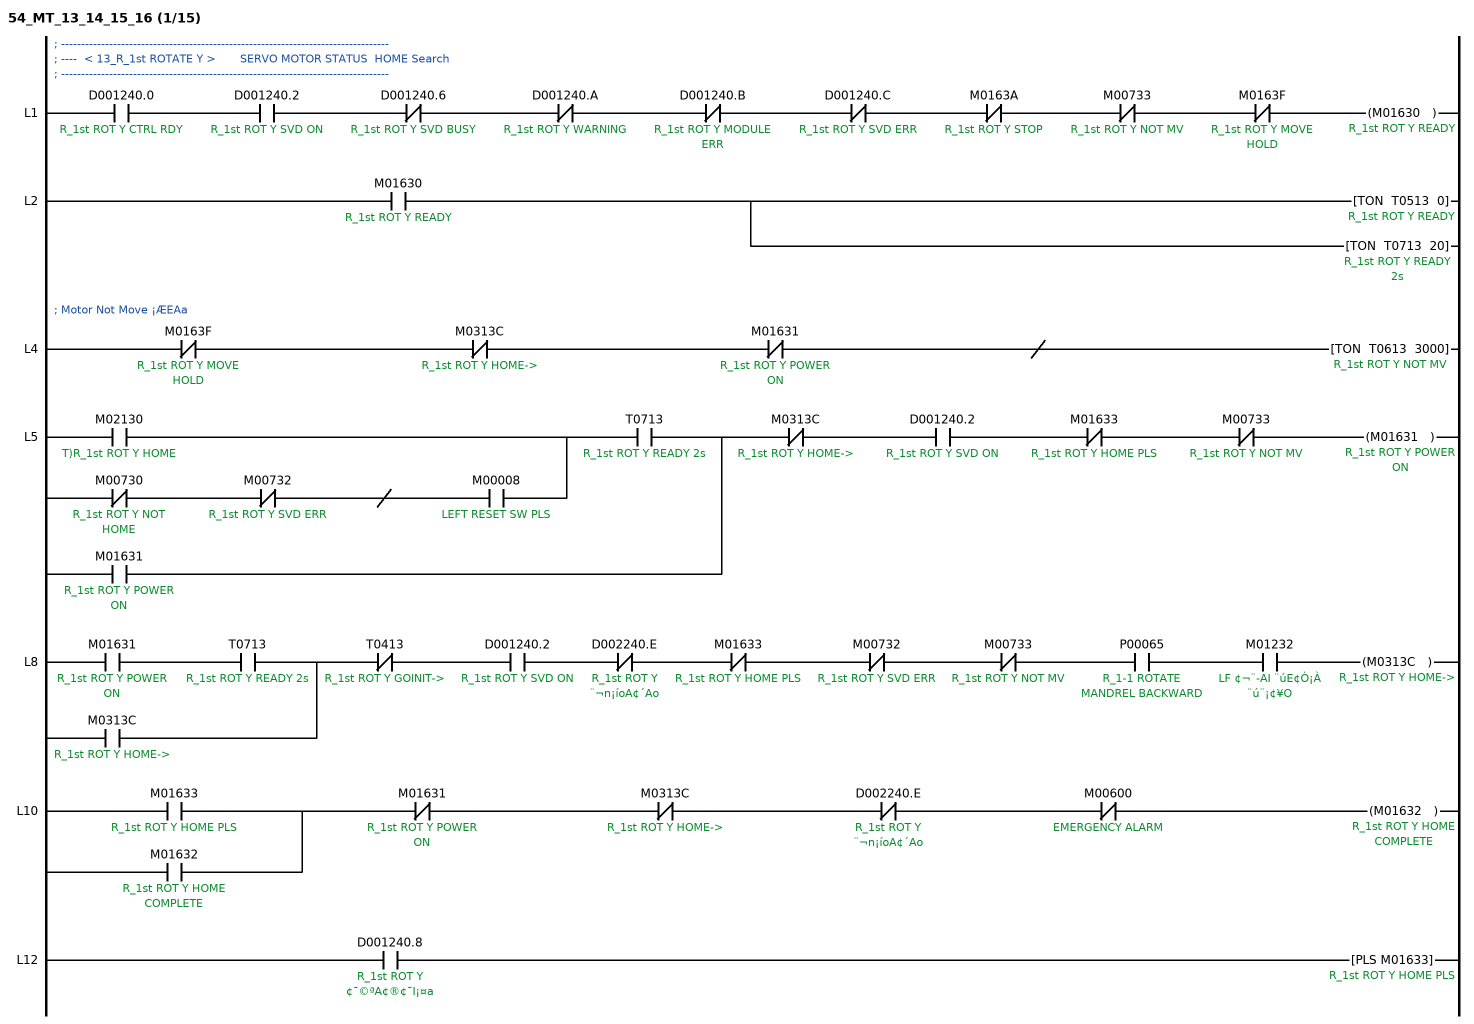
[picture p288: 54_MT_13_14_15_16 rungs L1-L12]
// ----------------------------------------------------------------------------------
// 
// ----  < 13_R_1st ROTATE Y >       SERVO MOTOR STATUS  HOME Search
// 
// ----------------------------------------------------------------------------------
; L1
LOAD      D001240.0	// R_1st ROT Y CTRL RDY
AND       D001240.2	// R_1st ROT Y SVD ON
AND NOT   D001240.6	// R_1st ROT Y SVD BUSY
AND NOT   D001240.A	// R_1st ROT Y WARNING
AND NOT   D001240.B	// R_1st ROT Y MODULE ERR
AND NOT   D001240.C	// R_1st ROT Y SVD ERR
AND NOT   M0163A	// R_1st ROT Y STOP
AND NOT   M00733	// R_1st ROT Y NOT MV
AND NOT   M0163F	// R_1st ROT Y MOVE HOLD
OUT       M01630	// R_1st ROT Y READY
; L2
LOAD      M01630	// R_1st ROT Y READY
TON       T0513 0	// R_1st ROT Y READY
TON       T0713 20	// R_1st ROT Y READY 2s
; L4
LOAD NOT  M0163F	// R_1st ROT Y MOVE HOLD
AND NOT   M0313C	// R_1st ROT Y HOME->
AND NOT   M01631	// R_1st ROT Y POWER ON
NOT
TON       T0613 3000	// R_1st ROT Y NOT MV
// output comment: Motor Not Move ¡ÆEAa
; L5
LOAD      M02130	// T)R_1st ROT Y HOME
LOAD NOT  M00730	// R_1st ROT Y NOT HOME
AND NOT   M00732	// R_1st ROT Y SVD ERR
NOT
AND       M00008	// LEFT RESET SW PLS
OR LOAD
AND       T0713	// R_1st ROT Y READY 2s
OR        M01631	// R_1st ROT Y POWER ON
AND NOT   M0313C	// R_1st ROT Y HOME->
AND       D001240.2	// R_1st ROT Y SVD ON
AND NOT   M01633	// R_1st ROT Y HOME PLS
AND NOT   M00733	// R_1st ROT Y NOT MV
OUT       M01631	// R_1st ROT Y POWER ON
; L8
LOAD      M01631	// R_1st ROT Y POWER ON
AND       T0713	// R_1st ROT Y READY 2s
OR        M0313C	// R_1st ROT Y HOME->
AND NOT   T0413	// R_1st ROT Y GOINIT->
AND       D001240.2	// R_1st ROT Y SVD ON
AND NOT   D002240.E	// R_1st ROT Y ¨¬n¡íoA¢´Ao
AND NOT   M01633	// R_1st ROT Y HOME PLS
AND NOT   M00732	// R_1st ROT Y SVD ERR
AND NOT   M00733	// R_1st ROT Y NOT MV
AND       P00065	// R_1-1 ROTATE MANDREL BACKWARD
AND       M01232	// LF ¢¬¨­AI ¨úE¢Ò¡À ¨ú¨¡¢¥O
OUT       M0313C	// R_1st ROT Y HOME->
; L10
LOAD      M01633	// R_1st ROT Y HOME PLS
OR        M01632	// R_1st ROT Y HOME COMPLETE
AND NOT   M01631	// R_1st ROT Y POWER ON
AND NOT   M0313C	// R_1st ROT Y HOME->
AND NOT   D002240.E	// R_1st ROT Y ¨¬n¡íoA¢´Ao
AND NOT   M00600	// EMERGENCY ALARM
OUT       M01632	// R_1st ROT Y HOME COMPLETE
; L12
LOAD      D001240.8	// R_1st ROT Y ¢¯©ªA¢®¢¯I¡¤a
OUTP      M01633	// R_1st ROT Y HOME PLS

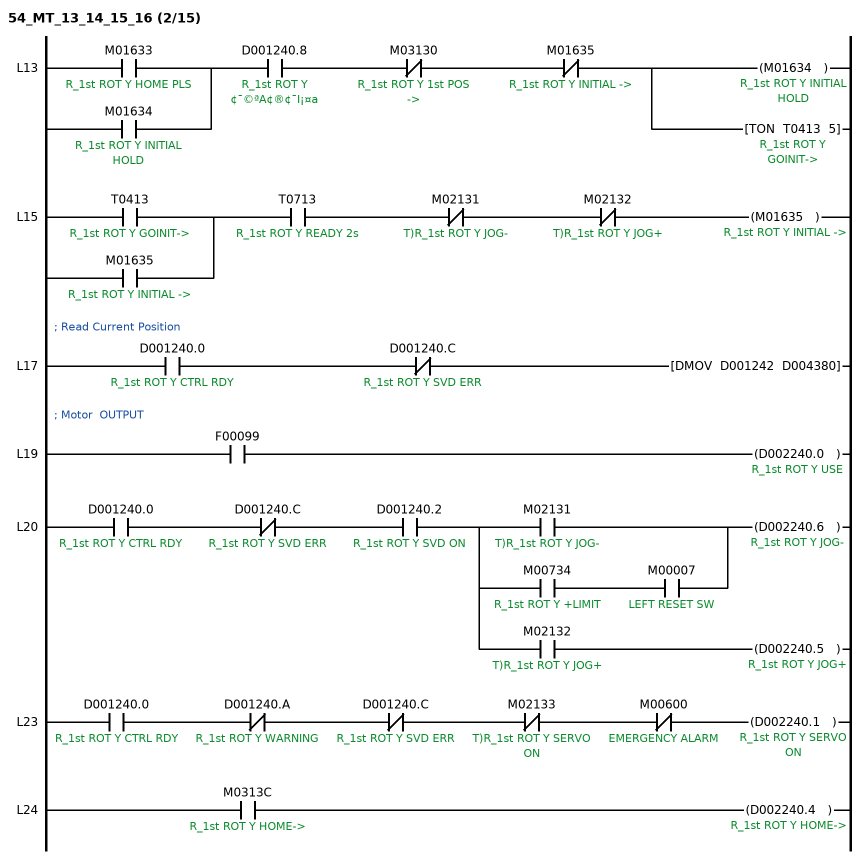
; L13
LOAD      M01633	// R_1st ROT Y HOME PLS
OR        M01634	// R_1st ROT Y INITIAL HOLD
AND       D001240.8	// R_1st ROT Y ¢¯©ªA¢®¢¯I¡¤a
AND NOT   M03130	// R_1st ROT Y 1st POS ->
AND NOT   M01635	// R_1st ROT Y INITIAL ->
OUT       M01634	// R_1st ROT Y INITIAL HOLD
TON       T0413 5	// R_1st ROT Y GOINIT->
; L15
LOAD      T0413	// R_1st ROT Y GOINIT->
OR        M01635	// R_1st ROT Y INITIAL ->
AND       T0713	// R_1st ROT Y READY 2s
AND NOT   M02131	// T)R_1st ROT Y JOG-
AND NOT   M02132	// T)R_1st ROT Y JOG+
OUT       M01635	// R_1st ROT Y INITIAL ->
; L17
LOAD      D001240.0	// R_1st ROT Y CTRL RDY
AND NOT   D001240.C	// R_1st ROT Y SVD ERR
DMOV      D001242 D004380
// output comment: Read Current Position
//  Motor  OUTPUT
; L19
LOAD      F00099
OUT       D002240.0	// R_1st ROT Y USE
; L20
LOAD      D001240.0	// R_1st ROT Y CTRL RDY
AND NOT   D001240.C	// R_1st ROT Y SVD ERR
AND       D001240.2	// R_1st ROT Y SVD ON
MPUSH
LOAD      M02131	// T)R_1st ROT Y JOG-
LOAD      M00734	// R_1st ROT Y +LIMIT
AND       M00007	// LEFT RESET SW
OR LOAD
AND LOAD
OUT       D002240.6	// R_1st ROT Y JOG-
MPOP
AND       M02132	// T)R_1st ROT Y JOG+
OUT       D002240.5	// R_1st ROT Y JOG+
; L23
LOAD      D001240.0	// R_1st ROT Y CTRL RDY
AND NOT   D001240.A	// R_1st ROT Y WARNING
AND NOT   D001240.C	// R_1st ROT Y SVD ERR
AND NOT   M02133	// T)R_1st ROT Y SERVO ON
AND NOT   M00600	// EMERGENCY ALARM
OUT       D002240.1	// R_1st ROT Y SERVO ON
; L24
LOAD      M0313C	// R_1st ROT Y HOME->
OUT       D002240.4	// R_1st ROT Y HOME->

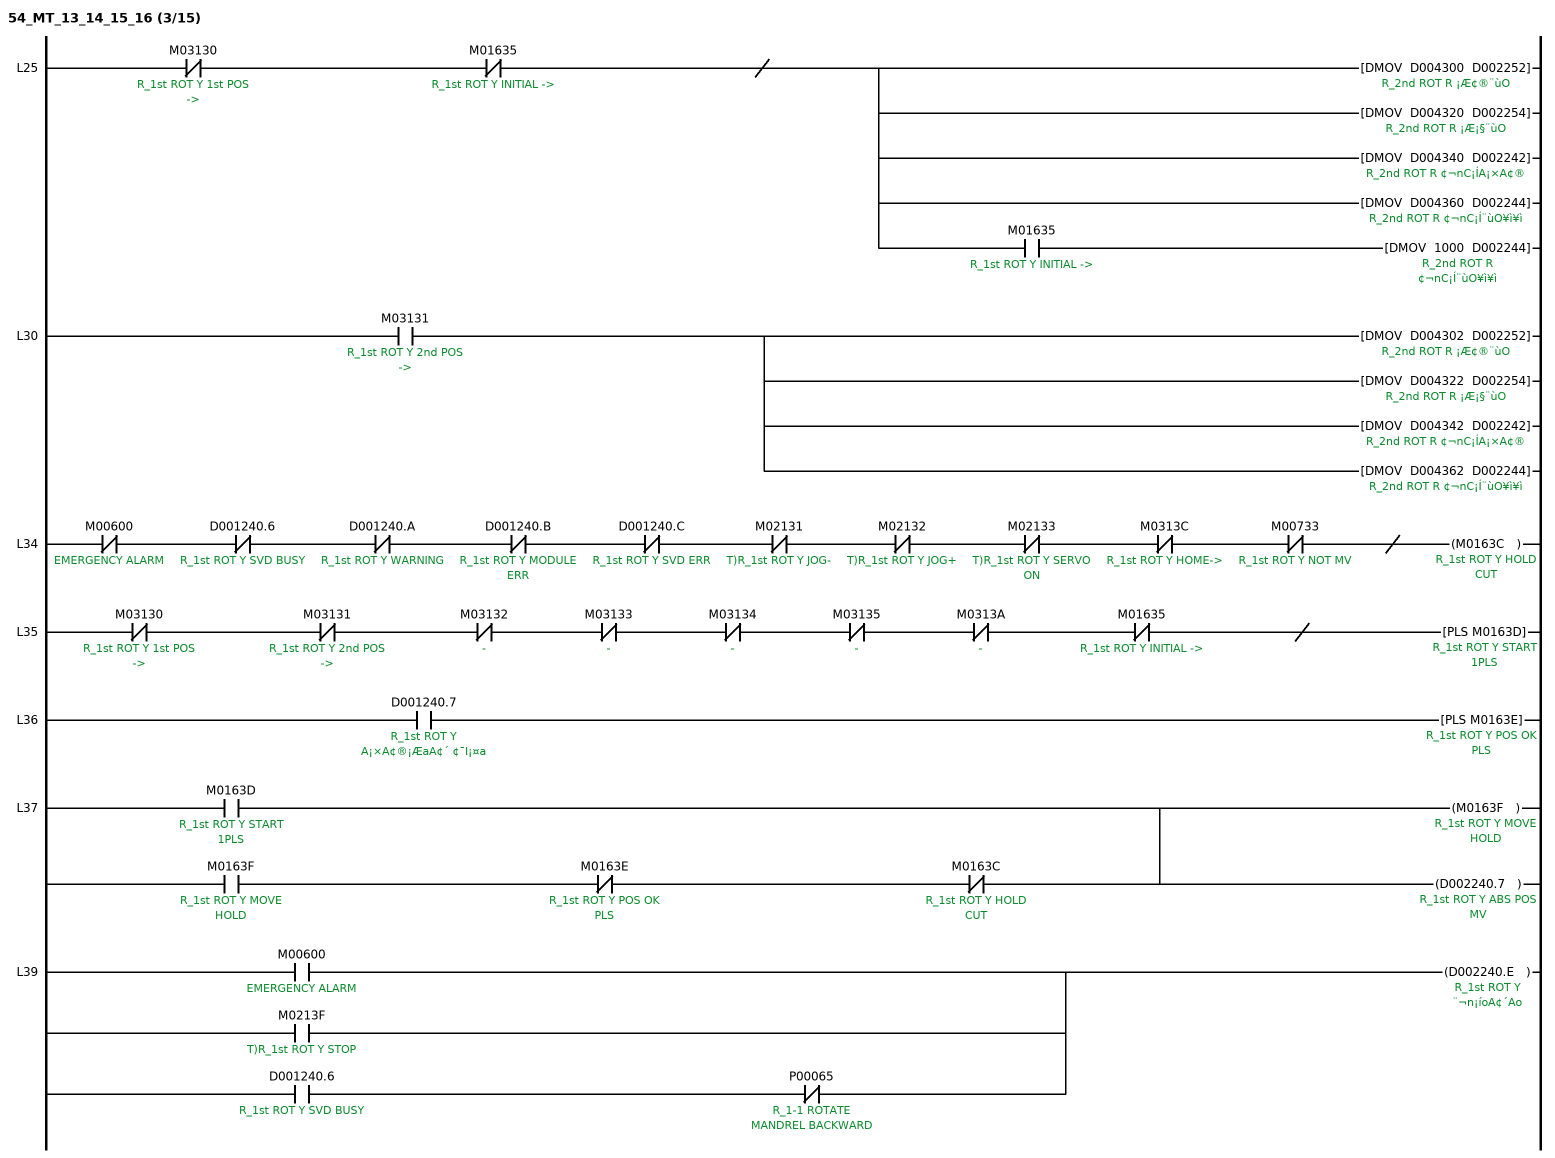
; L25
LOAD NOT  M03130	// R_1st ROT Y 1st POS ->
AND NOT   M01635	// R_1st ROT Y INITIAL ->
NOT
DMOV      D004300 D002252	// R_2nd ROT R ¡Æ¢®¨ùO
DMOV      D004320 D002254	// R_2nd ROT R ¡Æ¡§¨ùO
DMOV      D004340 D002242	// R_2nd ROT R ¢¬nC¡ÍA¡×A¢®
DMOV      D004360 D002244	// R_2nd ROT R ¢¬nC¡Í¨ùO¥ì¥ì
AND       M01635	// R_1st ROT Y INITIAL ->
DMOV      1000 D002244	// R_2nd ROT R ¢¬nC¡Í¨ùO¥ì¥ì
; L30
LOAD      M03131	// R_1st ROT Y 2nd POS ->
DMOV      D004302 D002252	// R_2nd ROT R ¡Æ¢®¨ùO
DMOV      D004322 D002254	// R_2nd ROT R ¡Æ¡§¨ùO
DMOV      D004342 D002242	// R_2nd ROT R ¢¬nC¡ÍA¡×A¢®
DMOV      D004362 D002244	// R_2nd ROT R ¢¬nC¡Í¨ùO¥ì¥ì
; L34
LOAD NOT  M00600	// EMERGENCY ALARM
AND NOT   D001240.6	// R_1st ROT Y SVD BUSY
AND NOT   D001240.A	// R_1st ROT Y WARNING
AND NOT   D001240.B	// R_1st ROT Y MODULE ERR
AND NOT   D001240.C	// R_1st ROT Y SVD ERR
AND NOT   M02131	// T)R_1st ROT Y JOG-
AND NOT   M02132	// T)R_1st ROT Y JOG+
AND NOT   M02133	// T)R_1st ROT Y SERVO ON
AND NOT   M0313C	// R_1st ROT Y HOME->
AND NOT   M00733	// R_1st ROT Y NOT MV
NOT
OUT       M0163C	// R_1st ROT Y HOLD CUT
; L35
LOAD NOT  M03130	// R_1st ROT Y 1st POS ->
AND NOT   M03131	// R_1st ROT Y 2nd POS ->
AND NOT   M03132	// -
AND NOT   M03133	// -
AND NOT   M03134	// -
AND NOT   M03135	// -
AND NOT   M0313A	// -
AND NOT   M01635	// R_1st ROT Y INITIAL ->
NOT
OUTP      M0163D	// R_1st ROT Y START 1PLS
; L36
LOAD      D001240.7	// R_1st ROT Y A¡×A¢®¡ÆaA¢´ ¢¯I¡¤a
OUTP      M0163E	// R_1st ROT Y POS OK PLS
; L37
LOAD      M0163D	// R_1st ROT Y START 1PLS
LOAD      M0163F	// R_1st ROT Y MOVE HOLD
AND NOT   M0163E	// R_1st ROT Y POS OK PLS
AND NOT   M0163C	// R_1st ROT Y HOLD CUT
OR LOAD
OUT       M0163F	// R_1st ROT Y MOVE HOLD
OUT       D002240.7	// R_1st ROT Y ABS POS MV
; L39
LOAD      M00600	// EMERGENCY ALARM
OR        M0213F	// T)R_1st ROT Y STOP
LOAD      D001240.6	// R_1st ROT Y SVD BUSY
AND NOT   P00065	// R_1-1 ROTATE MANDREL BACKWARD
OR LOAD
OUT       D002240.E	// R_1st ROT Y ¨¬n¡íoA¢´Ao

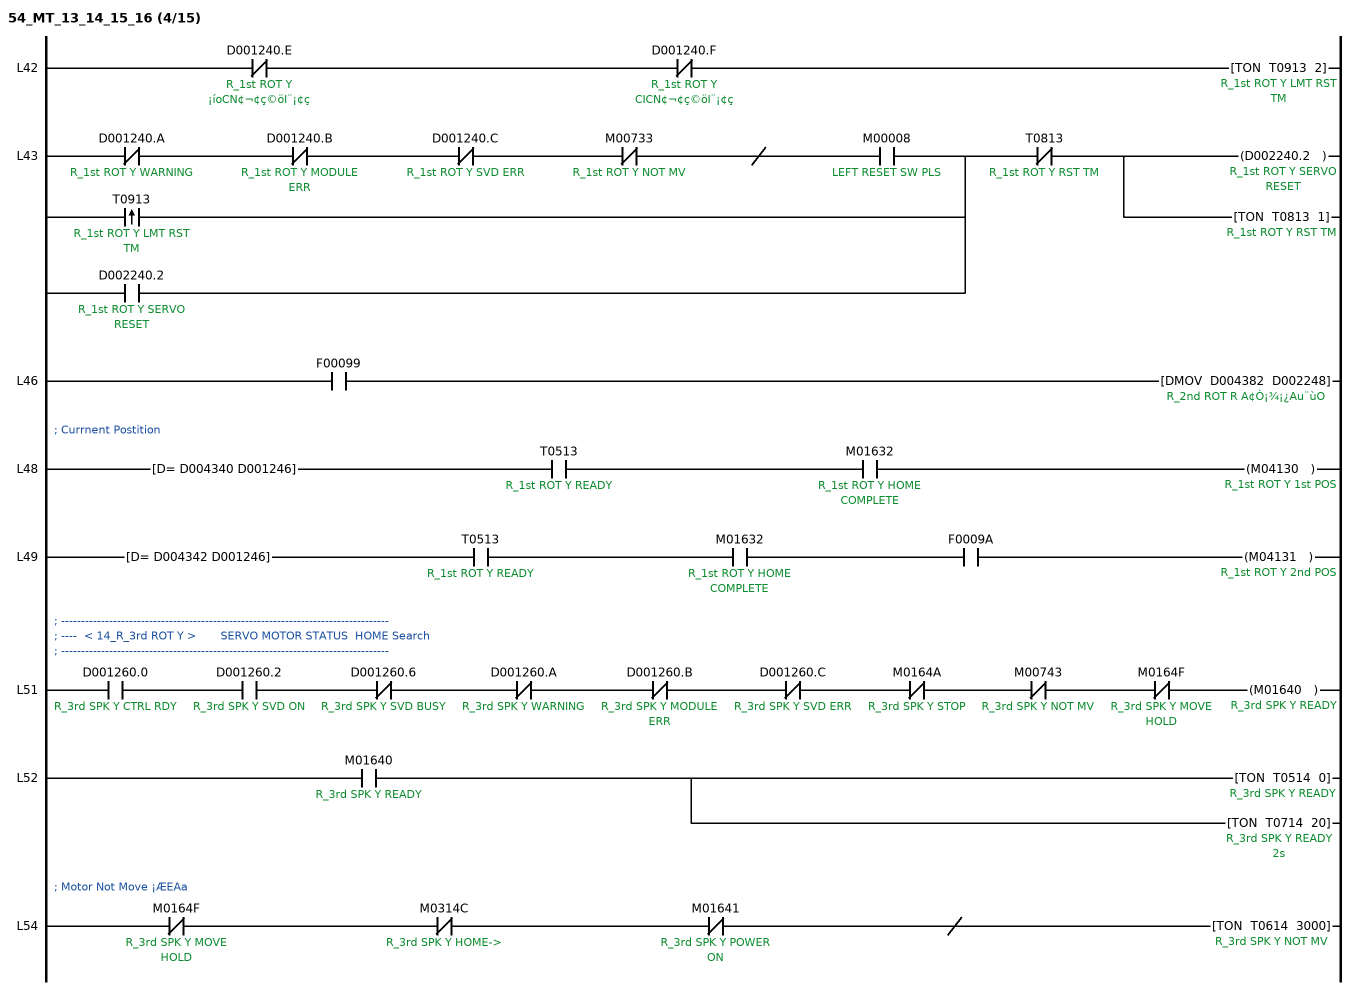
; L42
LOAD NOT  D001240.E	// R_1st ROT Y ¡íoCN¢¬¢ç©öI¨¡¢ç
AND NOT   D001240.F	// R_1st ROT Y CICN¢¬¢ç©öI¨¡¢ç
TON       T0913 2	// R_1st ROT Y LMT RST TM
; L43
LOAD NOT  D001240.A	// R_1st ROT Y WARNING
AND NOT   D001240.B	// R_1st ROT Y MODULE ERR
AND NOT   D001240.C	// R_1st ROT Y SVD ERR
AND NOT   M00733	// R_1st ROT Y NOT MV
NOT
AND       M00008	// LEFT RESET SW PLS
ORP       T0913	// R_1st ROT Y LMT RST TM
OR        D002240.2	// R_1st ROT Y SERVO RESET
AND NOT   T0813	// R_1st ROT Y RST TM
OUT       D002240.2	// R_1st ROT Y SERVO RESET
TON       T0813 1	// R_1st ROT Y RST TM
; L46
LOAD      F00099
DMOV      D004382 D002248	// R_2nd ROT R A¢Ò¡¾¡¿Au¨ùO
// Currnent Postition
; L48
LOADD=    D004340 D001246
AND       T0513	// R_1st ROT Y READY
AND       M01632	// R_1st ROT Y HOME COMPLETE
OUT       M04130	// R_1st ROT Y 1st POS
; L49
LOADD=    D004342 D001246
AND       T0513	// R_1st ROT Y READY
AND       M01632	// R_1st ROT Y HOME COMPLETE
AND       F0009A
OUT       M04131	// R_1st ROT Y 2nd POS
// ----------------------------------------------------------------------------------
// 
// ----  < 14_R_3rd ROT Y >       SERVO MOTOR STATUS  HOME Search
// 
// ----------------------------------------------------------------------------------
; L51
LOAD      D001260.0	// R_3rd SPK Y CTRL RDY
AND       D001260.2	// R_3rd SPK Y SVD ON
AND NOT   D001260.6	// R_3rd SPK Y SVD BUSY
AND NOT   D001260.A	// R_3rd SPK Y WARNING
AND NOT   D001260.B	// R_3rd SPK Y MODULE ERR
AND NOT   D001260.C	// R_3rd SPK Y SVD ERR
AND NOT   M0164A	// R_3rd SPK Y STOP
AND NOT   M00743	// R_3rd SPK Y NOT MV
AND NOT   M0164F	// R_3rd SPK Y MOVE HOLD
OUT       M01640	// R_3rd SPK Y READY
; L52
LOAD      M01640	// R_3rd SPK Y READY
TON       T0514 0	// R_3rd SPK Y READY
TON       T0714 20	// R_3rd SPK Y READY 2s
; L54
LOAD NOT  M0164F	// R_3rd SPK Y MOVE HOLD
AND NOT   M0314C	// R_3rd SPK Y HOME->
AND NOT   M01641	// R_3rd SPK Y POWER ON
NOT
TON       T0614 3000	// R_3rd SPK Y NOT MV
// output comment: Motor Not Move ¡ÆEAa

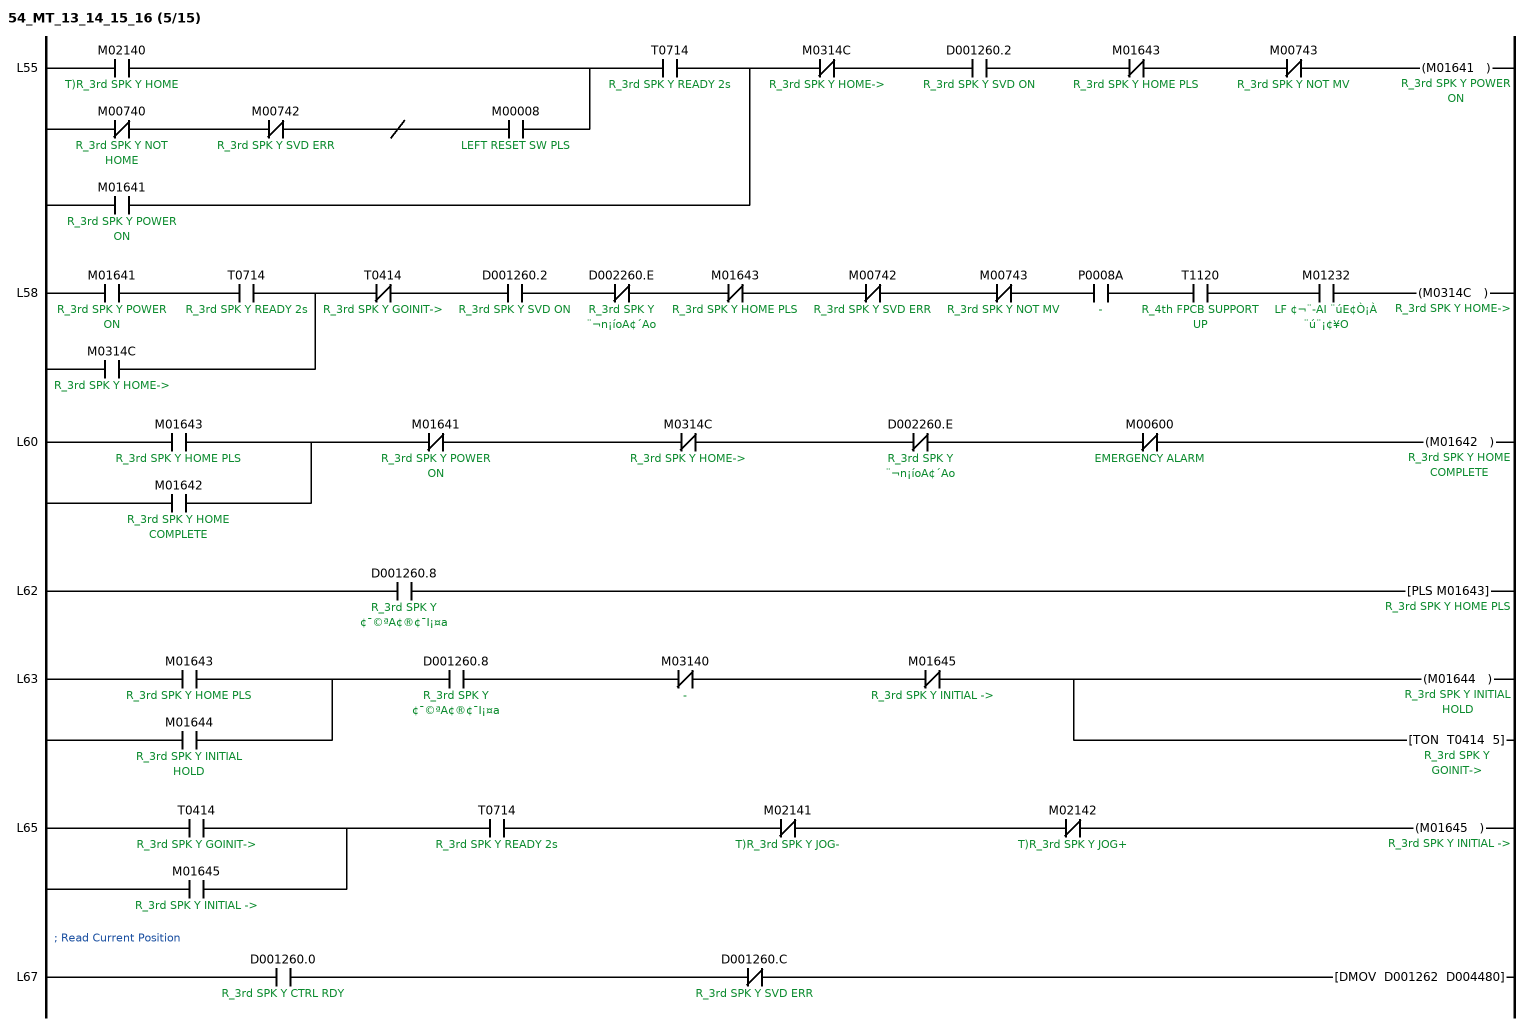
; L55
LOAD      M02140	// T)R_3rd SPK Y HOME
LOAD NOT  M00740	// R_3rd SPK Y NOT HOME
AND NOT   M00742	// R_3rd SPK Y SVD ERR
NOT
AND       M00008	// LEFT RESET SW PLS
OR LOAD
AND       T0714	// R_3rd SPK Y READY 2s
OR        M01641	// R_3rd SPK Y POWER ON
AND NOT   M0314C	// R_3rd SPK Y HOME->
AND       D001260.2	// R_3rd SPK Y SVD ON
AND NOT   M01643	// R_3rd SPK Y HOME PLS
AND NOT   M00743	// R_3rd SPK Y NOT MV
OUT       M01641	// R_3rd SPK Y POWER ON
; L58
LOAD      M01641	// R_3rd SPK Y POWER ON
AND       T0714	// R_3rd SPK Y READY 2s
OR        M0314C	// R_3rd SPK Y HOME->
AND NOT   T0414	// R_3rd SPK Y GOINIT->
AND       D001260.2	// R_3rd SPK Y SVD ON
AND NOT   D002260.E	// R_3rd SPK Y ¨¬n¡íoA¢´Ao
AND NOT   M01643	// R_3rd SPK Y HOME PLS
AND NOT   M00742	// R_3rd SPK Y SVD ERR
AND NOT   M00743	// R_3rd SPK Y NOT MV
AND       P0008A	// -
AND       T1120	// R_4th FPCB SUPPORT UP
AND       M01232	// LF ¢¬¨­AI ¨úE¢Ò¡À ¨ú¨¡¢¥O
OUT       M0314C	// R_3rd SPK Y HOME->
; L60
LOAD      M01643	// R_3rd SPK Y HOME PLS
OR        M01642	// R_3rd SPK Y HOME COMPLETE
AND NOT   M01641	// R_3rd SPK Y POWER ON
AND NOT   M0314C	// R_3rd SPK Y HOME->
AND NOT   D002260.E	// R_3rd SPK Y ¨¬n¡íoA¢´Ao
AND NOT   M00600	// EMERGENCY ALARM
OUT       M01642	// R_3rd SPK Y HOME COMPLETE
; L62
LOAD      D001260.8	// R_3rd SPK Y ¢¯©ªA¢®¢¯I¡¤a
OUTP      M01643	// R_3rd SPK Y HOME PLS
; L63
LOAD      M01643	// R_3rd SPK Y HOME PLS
OR        M01644	// R_3rd SPK Y INITIAL HOLD
AND       D001260.8	// R_3rd SPK Y ¢¯©ªA¢®¢¯I¡¤a
AND NOT   M03140	// -
AND NOT   M01645	// R_3rd SPK Y INITIAL ->
OUT       M01644	// R_3rd SPK Y INITIAL HOLD
TON       T0414 5	// R_3rd SPK Y GOINIT->
; L65
LOAD      T0414	// R_3rd SPK Y GOINIT->
OR        M01645	// R_3rd SPK Y INITIAL ->
AND       T0714	// R_3rd SPK Y READY 2s
AND NOT   M02141	// T)R_3rd SPK Y JOG-
AND NOT   M02142	// T)R_3rd SPK Y JOG+
OUT       M01645	// R_3rd SPK Y INITIAL ->
; L67
LOAD      D001260.0	// R_3rd SPK Y CTRL RDY
AND NOT   D001260.C	// R_3rd SPK Y SVD ERR
DMOV      D001262 D004480
// output comment: Read Current Position

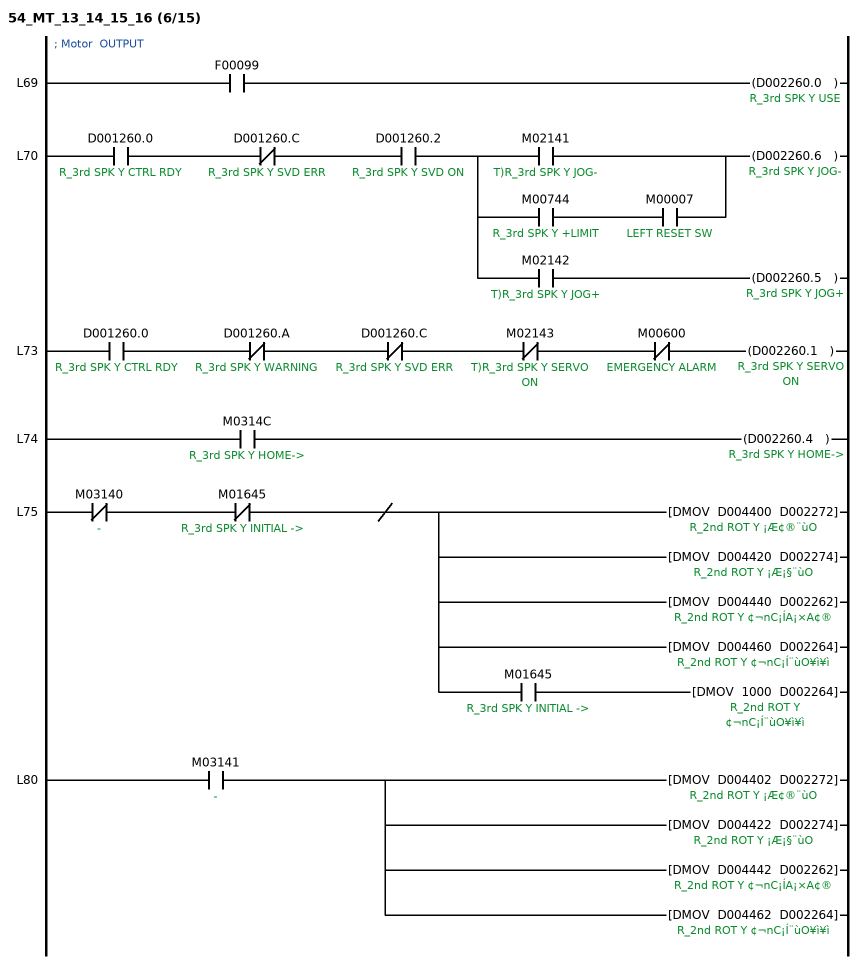
//  Motor  OUTPUT
; L69
LOAD      F00099
OUT       D002260.0	// R_3rd SPK Y USE
; L70
LOAD      D001260.0	// R_3rd SPK Y CTRL RDY
AND NOT   D001260.C	// R_3rd SPK Y SVD ERR
AND       D001260.2	// R_3rd SPK Y SVD ON
MPUSH
LOAD      M02141	// T)R_3rd SPK Y JOG-
LOAD      M00744	// R_3rd SPK Y +LIMIT
AND       M00007	// LEFT RESET SW
OR LOAD
AND LOAD
OUT       D002260.6	// R_3rd SPK Y JOG-
MPOP
AND       M02142	// T)R_3rd SPK Y JOG+
OUT       D002260.5	// R_3rd SPK Y JOG+
; L73
LOAD      D001260.0	// R_3rd SPK Y CTRL RDY
AND NOT   D001260.A	// R_3rd SPK Y WARNING
AND NOT   D001260.C	// R_3rd SPK Y SVD ERR
AND NOT   M02143	// T)R_3rd SPK Y SERVO ON
AND NOT   M00600	// EMERGENCY ALARM
OUT       D002260.1	// R_3rd SPK Y SERVO ON
; L74
LOAD      M0314C	// R_3rd SPK Y HOME->
OUT       D002260.4	// R_3rd SPK Y HOME->
; L75
LOAD NOT  M03140	// -
AND NOT   M01645	// R_3rd SPK Y INITIAL ->
NOT
DMOV      D004400 D002272	// R_2nd ROT Y ¡Æ¢®¨ùO
DMOV      D004420 D002274	// R_2nd ROT Y ¡Æ¡§¨ùO
DMOV      D004440 D002262	// R_2nd ROT Y ¢¬nC¡ÍA¡×A¢®
DMOV      D004460 D002264	// R_2nd ROT Y ¢¬nC¡Í¨ùO¥ì¥ì
AND       M01645	// R_3rd SPK Y INITIAL ->
DMOV      1000 D002264	// R_2nd ROT Y ¢¬nC¡Í¨ùO¥ì¥ì
; L80
LOAD      M03141	// -
DMOV      D004402 D002272	// R_2nd ROT Y ¡Æ¢®¨ùO
DMOV      D004422 D002274	// R_2nd ROT Y ¡Æ¡§¨ùO
DMOV      D004442 D002262	// R_2nd ROT Y ¢¬nC¡ÍA¡×A¢®
DMOV      D004462 D002264	// R_2nd ROT Y ¢¬nC¡Í¨ùO¥ì¥ì

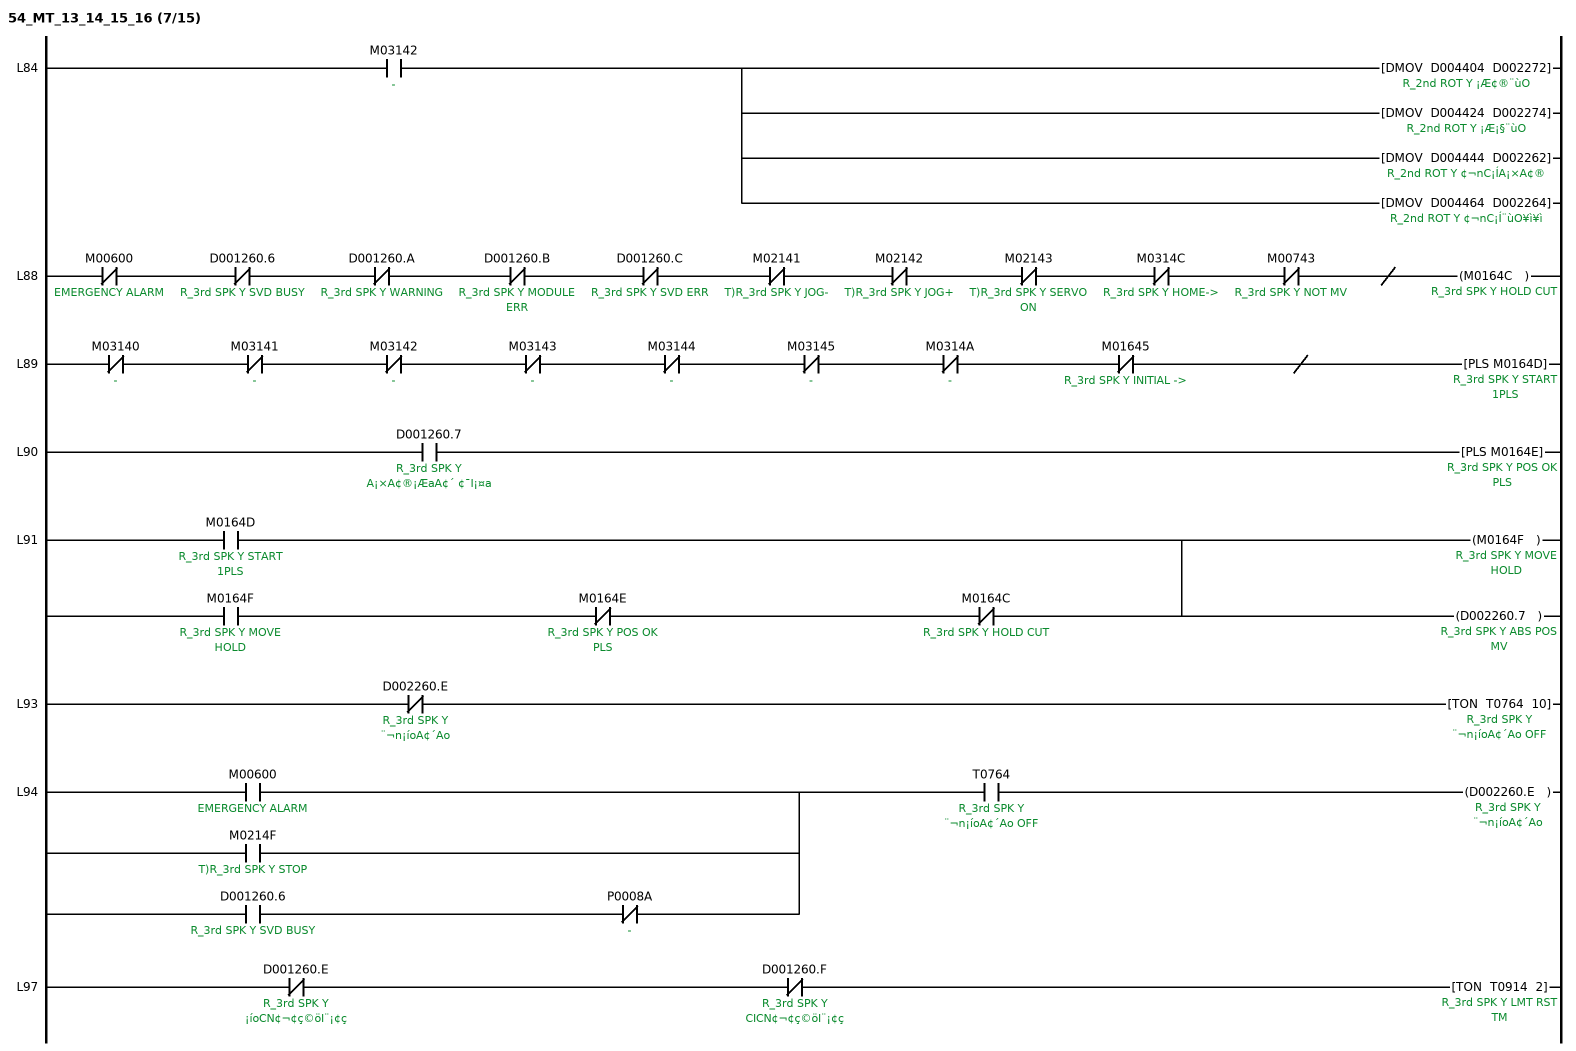
; L84
LOAD      M03142	// -
DMOV      D004404 D002272	// R_2nd ROT Y ¡Æ¢®¨ùO
DMOV      D004424 D002274	// R_2nd ROT Y ¡Æ¡§¨ùO
DMOV      D004444 D002262	// R_2nd ROT Y ¢¬nC¡ÍA¡×A¢®
DMOV      D004464 D002264	// R_2nd ROT Y ¢¬nC¡Í¨ùO¥ì¥ì
; L88
LOAD NOT  M00600	// EMERGENCY ALARM
AND NOT   D001260.6	// R_3rd SPK Y SVD BUSY
AND NOT   D001260.A	// R_3rd SPK Y WARNING
AND NOT   D001260.B	// R_3rd SPK Y MODULE ERR
AND NOT   D001260.C	// R_3rd SPK Y SVD ERR
AND NOT   M02141	// T)R_3rd SPK Y JOG-
AND NOT   M02142	// T)R_3rd SPK Y JOG+
AND NOT   M02143	// T)R_3rd SPK Y SERVO ON
AND NOT   M0314C	// R_3rd SPK Y HOME->
AND NOT   M00743	// R_3rd SPK Y NOT MV
NOT
OUT       M0164C	// R_3rd SPK Y HOLD CUT
; L89
LOAD NOT  M03140	// -
AND NOT   M03141	// -
AND NOT   M03142	// -
AND NOT   M03143	// -
AND NOT   M03144	// -
AND NOT   M03145	// -
AND NOT   M0314A	// -
AND NOT   M01645	// R_3rd SPK Y INITIAL ->
NOT
OUTP      M0164D	// R_3rd SPK Y START 1PLS
; L90
LOAD      D001260.7	// R_3rd SPK Y A¡×A¢®¡ÆaA¢´ ¢¯I¡¤a
OUTP      M0164E	// R_3rd SPK Y POS OK PLS
; L91
LOAD      M0164D	// R_3rd SPK Y START 1PLS
LOAD      M0164F	// R_3rd SPK Y MOVE HOLD
AND NOT   M0164E	// R_3rd SPK Y POS OK PLS
AND NOT   M0164C	// R_3rd SPK Y HOLD CUT
OR LOAD
OUT       M0164F	// R_3rd SPK Y MOVE HOLD
OUT       D002260.7	// R_3rd SPK Y ABS POS MV
; L93
LOAD NOT  D002260.E	// R_3rd SPK Y ¨¬n¡íoA¢´Ao
TON       T0764 10	// R_3rd SPK Y ¨¬n¡íoA¢´Ao OFF
; L94
LOAD      M00600	// EMERGENCY ALARM
OR        M0214F	// T)R_3rd SPK Y STOP
LOAD      D001260.6	// R_3rd SPK Y SVD BUSY
AND NOT   P0008A	// -
OR LOAD
AND       T0764	// R_3rd SPK Y ¨¬n¡íoA¢´Ao OFF
OUT       D002260.E	// R_3rd SPK Y ¨¬n¡íoA¢´Ao
; L97
LOAD NOT  D001260.E	// R_3rd SPK Y ¡íoCN¢¬¢ç©öI¨¡¢ç
AND NOT   D001260.F	// R_3rd SPK Y CICN¢¬¢ç©öI¨¡¢ç
TON       T0914 2	// R_3rd SPK Y LMT RST TM

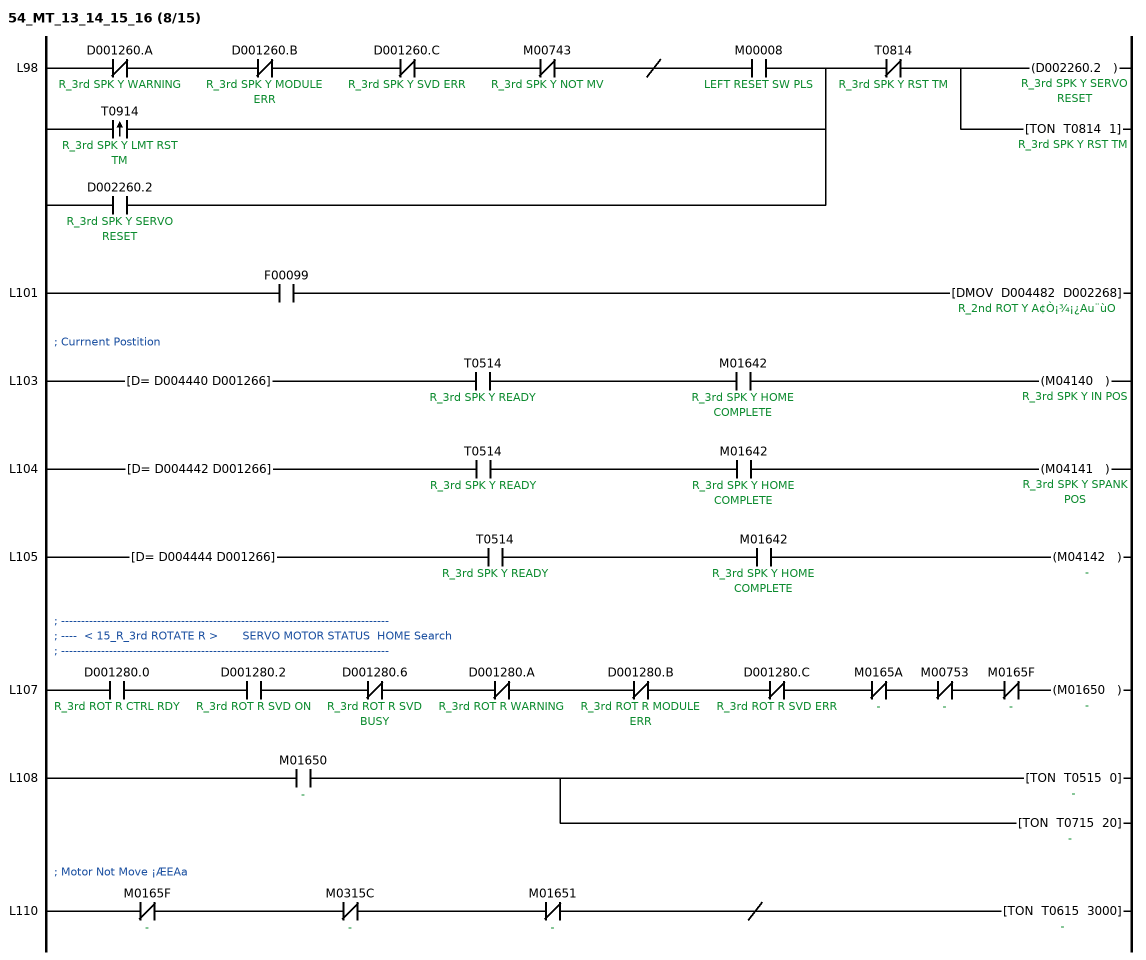
; L98
LOAD NOT  D001260.A	// R_3rd SPK Y WARNING
AND NOT   D001260.B	// R_3rd SPK Y MODULE ERR
AND NOT   D001260.C	// R_3rd SPK Y SVD ERR
AND NOT   M00743	// R_3rd SPK Y NOT MV
NOT
AND       M00008	// LEFT RESET SW PLS
ORP       T0914	// R_3rd SPK Y LMT RST TM
OR        D002260.2	// R_3rd SPK Y SERVO RESET
AND NOT   T0814	// R_3rd SPK Y RST TM
OUT       D002260.2	// R_3rd SPK Y SERVO RESET
TON       T0814 1	// R_3rd SPK Y RST TM
; L101
LOAD      F00099
DMOV      D004482 D002268	// R_2nd ROT Y A¢Ò¡¾¡¿Au¨ùO
// Currnent Postition
; L103
LOADD=    D004440 D001266
AND       T0514	// R_3rd SPK Y READY
AND       M01642	// R_3rd SPK Y HOME COMPLETE
OUT       M04140	// R_3rd SPK Y IN POS
; L104
LOADD=    D004442 D001266
AND       T0514	// R_3rd SPK Y READY
AND       M01642	// R_3rd SPK Y HOME COMPLETE
OUT       M04141	// R_3rd SPK Y SPANK POS
; L105
LOADD=    D004444 D001266
AND       T0514	// R_3rd SPK Y READY
AND       M01642	// R_3rd SPK Y HOME COMPLETE
OUT       M04142	// -
// ----------------------------------------------------------------------------------
// 
// ----  < 15_R_3rd ROTATE R >       SERVO MOTOR STATUS  HOME Search
// 
// ----------------------------------------------------------------------------------
; L107
LOAD      D001280.0	// R_3rd ROT R CTRL RDY
AND       D001280.2	// R_3rd ROT R SVD ON
AND NOT   D001280.6	// R_3rd ROT R SVD BUSY
AND NOT   D001280.A	// R_3rd ROT R WARNING
AND NOT   D001280.B	// R_3rd ROT R MODULE ERR
AND NOT   D001280.C	// R_3rd ROT R SVD ERR
AND NOT   M0165A	// -
AND NOT   M00753	// -
AND NOT   M0165F	// -
OUT       M01650	// -
; L108
LOAD      M01650	// -
TON       T0515 0	// -
TON       T0715 20	// -
; L110
LOAD NOT  M0165F	// -
AND NOT   M0315C	// -
AND NOT   M01651	// -
NOT
TON       T0615 3000	// -
// output comment: Motor Not Move ¡ÆEAa

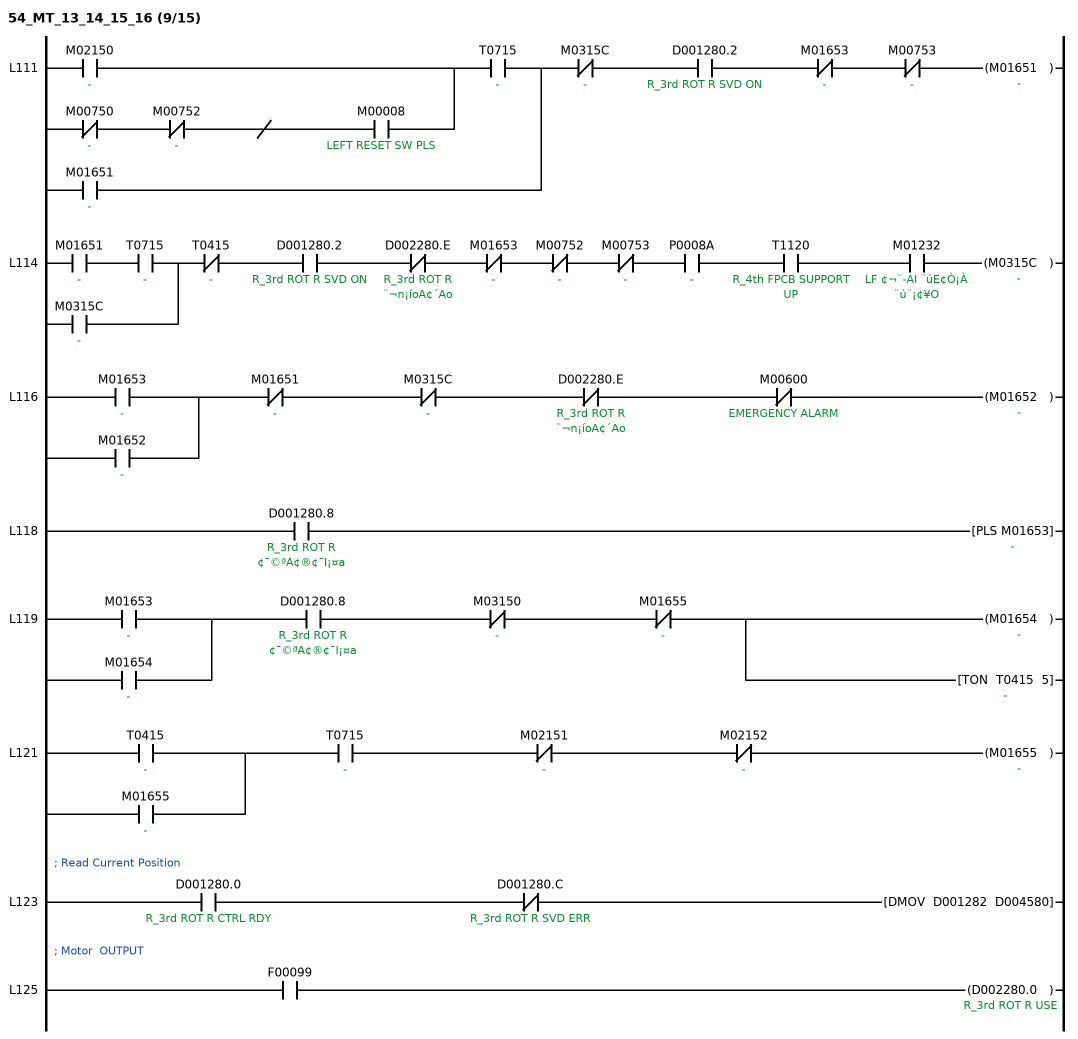
; L111
LOAD      M02150	// -
LOAD NOT  M00750	// -
AND NOT   M00752	// -
NOT
AND       M00008	// LEFT RESET SW PLS
OR LOAD
AND       T0715	// -
OR        M01651	// -
AND NOT   M0315C	// -
AND       D001280.2	// R_3rd ROT R SVD ON
AND NOT   M01653	// -
AND NOT   M00753	// -
OUT       M01651	// -
; L114
LOAD      M01651	// -
AND       T0715	// -
OR        M0315C	// -
AND NOT   T0415	// -
AND       D001280.2	// R_3rd ROT R SVD ON
AND NOT   D002280.E	// R_3rd ROT R ¨¬n¡íoA¢´Ao
AND NOT   M01653	// -
AND NOT   M00752	// -
AND NOT   M00753	// -
AND       P0008A	// -
AND       T1120	// R_4th FPCB SUPPORT UP
AND       M01232	// LF ¢¬¨­AI ¨úE¢Ò¡À ¨ú¨¡¢¥O
OUT       M0315C	// -
; L116
LOAD      M01653	// -
OR        M01652	// -
AND NOT   M01651	// -
AND NOT   M0315C	// -
AND NOT   D002280.E	// R_3rd ROT R ¨¬n¡íoA¢´Ao
AND NOT   M00600	// EMERGENCY ALARM
OUT       M01652	// -
; L118
LOAD      D001280.8	// R_3rd ROT R ¢¯©ªA¢®¢¯I¡¤a
OUTP      M01653	// -
; L119
LOAD      M01653	// -
OR        M01654	// -
AND       D001280.8	// R_3rd ROT R ¢¯©ªA¢®¢¯I¡¤a
AND NOT   M03150	// -
AND NOT   M01655	// -
OUT       M01654	// -
TON       T0415 5	// -
; L121
LOAD      T0415	// -
OR        M01655	// -
AND       T0715	// -
AND NOT   M02151	// -
AND NOT   M02152	// -
OUT       M01655	// -
; L123
LOAD      D001280.0	// R_3rd ROT R CTRL RDY
AND NOT   D001280.C	// R_3rd ROT R SVD ERR
DMOV      D001282 D004580
// output comment: Read Current Position
//  Motor  OUTPUT
; L125
LOAD      F00099
OUT       D002280.0	// R_3rd ROT R USE

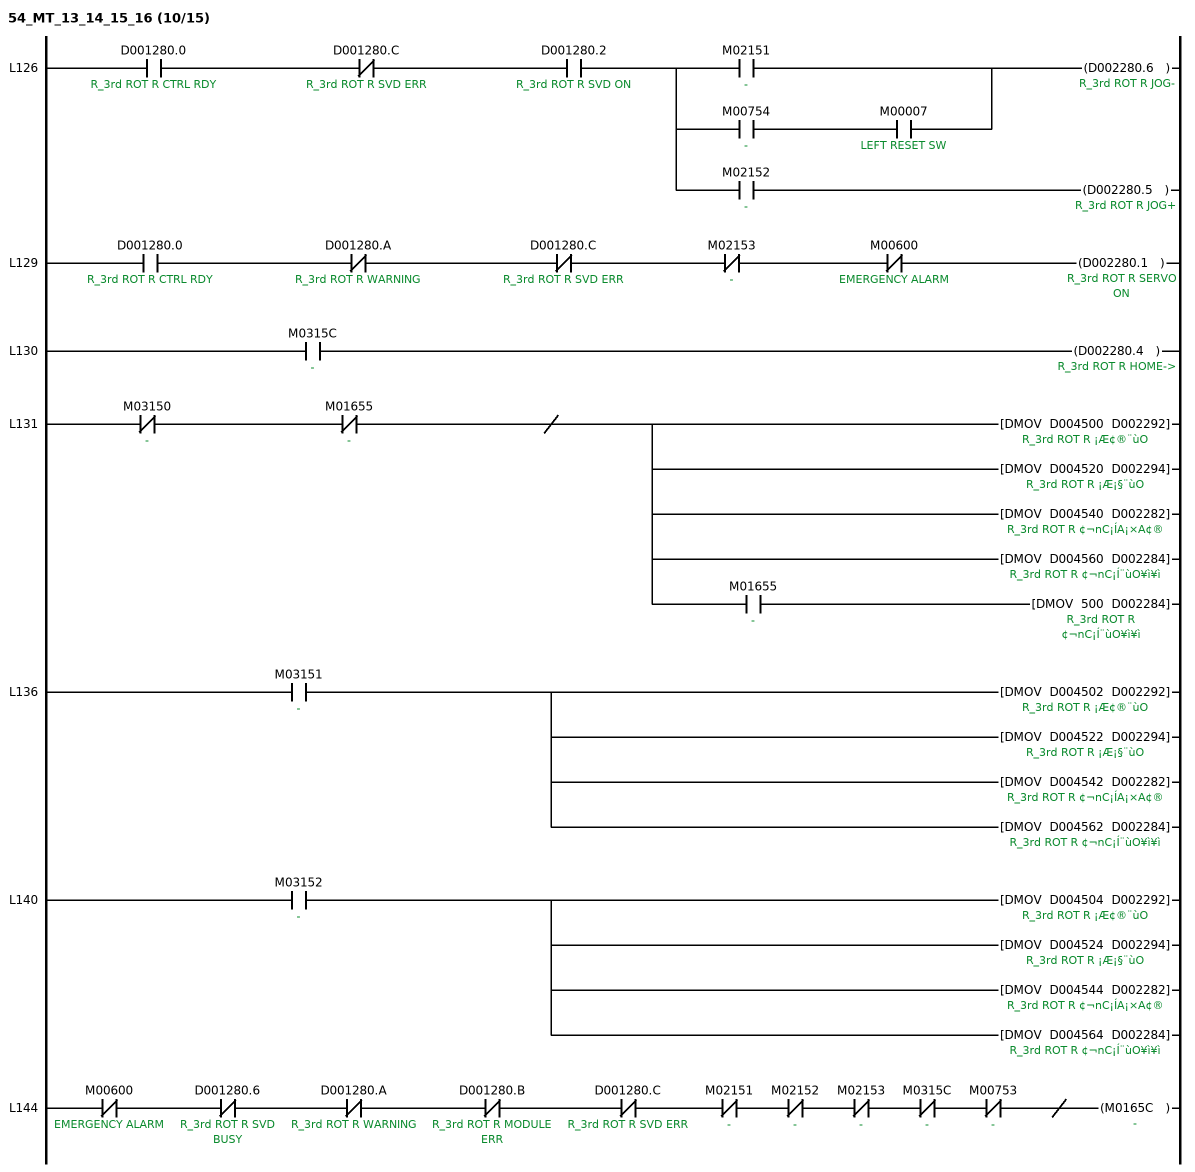
; L126
LOAD      D001280.0	// R_3rd ROT R CTRL RDY
AND NOT   D001280.C	// R_3rd ROT R SVD ERR
AND       D001280.2	// R_3rd ROT R SVD ON
MPUSH
LOAD      M02151	// -
LOAD      M00754	// -
AND       M00007	// LEFT RESET SW
OR LOAD
AND LOAD
OUT       D002280.6	// R_3rd ROT R JOG-
MPOP
AND       M02152	// -
OUT       D002280.5	// R_3rd ROT R JOG+
; L129
LOAD      D001280.0	// R_3rd ROT R CTRL RDY
AND NOT   D001280.A	// R_3rd ROT R WARNING
AND NOT   D001280.C	// R_3rd ROT R SVD ERR
AND NOT   M02153	// -
AND NOT   M00600	// EMERGENCY ALARM
OUT       D002280.1	// R_3rd ROT R SERVO ON
; L130
LOAD      M0315C	// -
OUT       D002280.4	// R_3rd ROT R HOME->
; L131
LOAD NOT  M03150	// -
AND NOT   M01655	// -
NOT
DMOV      D004500 D002292	// R_3rd ROT R ¡Æ¢®¨ùO
DMOV      D004520 D002294	// R_3rd ROT R ¡Æ¡§¨ùO
DMOV      D004540 D002282	// R_3rd ROT R ¢¬nC¡ÍA¡×A¢®
DMOV      D004560 D002284	// R_3rd ROT R ¢¬nC¡Í¨ùO¥ì¥ì
AND       M01655	// -
DMOV      500 D002284	// R_3rd ROT R ¢¬nC¡Í¨ùO¥ì¥ì
; L136
LOAD      M03151	// -
DMOV      D004502 D002292	// R_3rd ROT R ¡Æ¢®¨ùO
DMOV      D004522 D002294	// R_3rd ROT R ¡Æ¡§¨ùO
DMOV      D004542 D002282	// R_3rd ROT R ¢¬nC¡ÍA¡×A¢®
DMOV      D004562 D002284	// R_3rd ROT R ¢¬nC¡Í¨ùO¥ì¥ì
; L140
LOAD      M03152	// -
DMOV      D004504 D002292	// R_3rd ROT R ¡Æ¢®¨ùO
DMOV      D004524 D002294	// R_3rd ROT R ¡Æ¡§¨ùO
DMOV      D004544 D002282	// R_3rd ROT R ¢¬nC¡ÍA¡×A¢®
DMOV      D004564 D002284	// R_3rd ROT R ¢¬nC¡Í¨ùO¥ì¥ì
; L144
LOAD NOT  M00600	// EMERGENCY ALARM
AND NOT   D001280.6	// R_3rd ROT R SVD BUSY
AND NOT   D001280.A	// R_3rd ROT R WARNING
AND NOT   D001280.B	// R_3rd ROT R MODULE ERR
AND NOT   D001280.C	// R_3rd ROT R SVD ERR
AND NOT   M02151	// -
AND NOT   M02152	// -
AND NOT   M02153	// -
AND NOT   M0315C	// -
AND NOT   M00753	// -
NOT
OUT       M0165C	// -

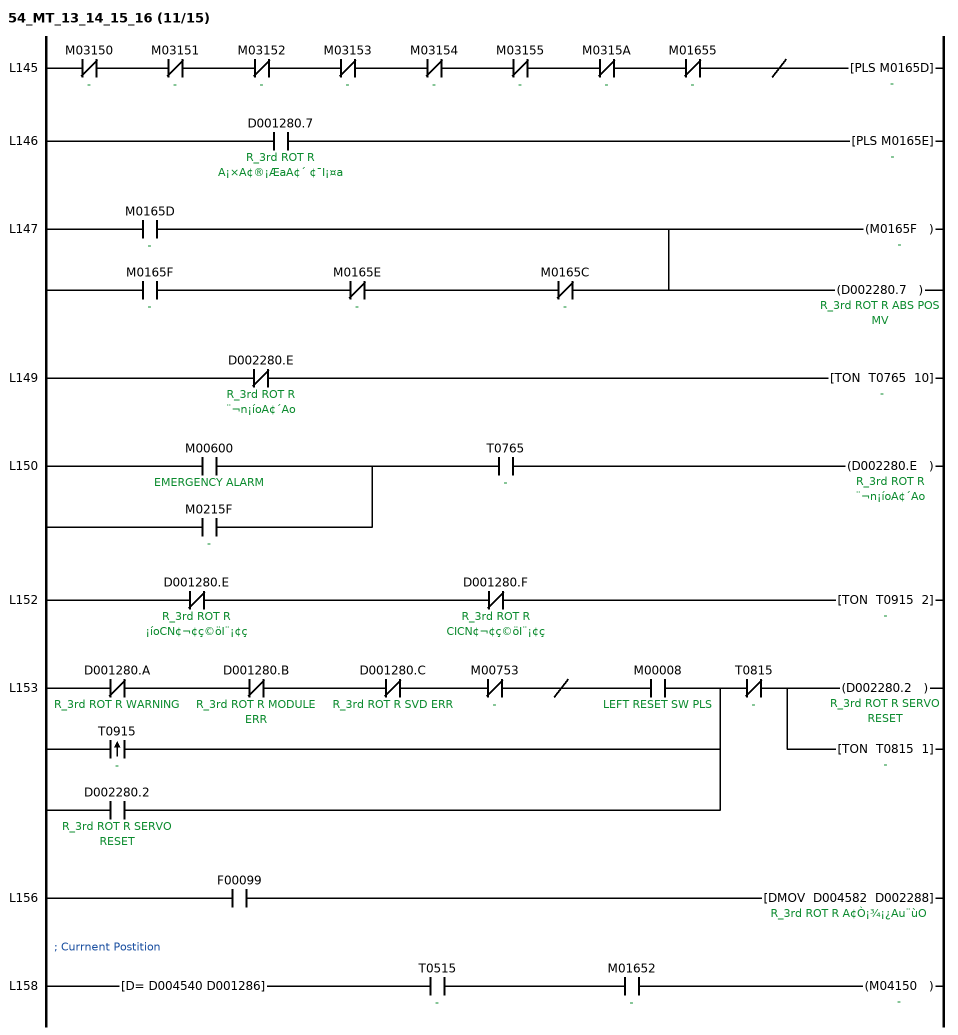
; L145
LOAD NOT  M03150	// -
AND NOT   M03151	// -
AND NOT   M03152	// -
AND NOT   M03153	// -
AND NOT   M03154	// -
AND NOT   M03155	// -
AND NOT   M0315A	// -
AND NOT   M01655	// -
NOT
OUTP      M0165D	// -
; L146
LOAD      D001280.7	// R_3rd ROT R A¡×A¢®¡ÆaA¢´ ¢¯I¡¤a
OUTP      M0165E	// -
; L147
LOAD      M0165D	// -
LOAD      M0165F	// -
AND NOT   M0165E	// -
AND NOT   M0165C	// -
OR LOAD
OUT       M0165F	// -
OUT       D002280.7	// R_3rd ROT R ABS POS MV
; L149
LOAD NOT  D002280.E	// R_3rd ROT R ¨¬n¡íoA¢´Ao
TON       T0765 10	// -
; L150
LOAD      M00600	// EMERGENCY ALARM
OR        M0215F	// -
AND       T0765	// -
OUT       D002280.E	// R_3rd ROT R ¨¬n¡íoA¢´Ao
; L152
LOAD NOT  D001280.E	// R_3rd ROT R ¡íoCN¢¬¢ç©öI¨¡¢ç
AND NOT   D001280.F	// R_3rd ROT R CICN¢¬¢ç©öI¨¡¢ç
TON       T0915 2	// -
; L153
LOAD NOT  D001280.A	// R_3rd ROT R WARNING
AND NOT   D001280.B	// R_3rd ROT R MODULE ERR
AND NOT   D001280.C	// R_3rd ROT R SVD ERR
AND NOT   M00753	// -
NOT
AND       M00008	// LEFT RESET SW PLS
ORP       T0915	// -
OR        D002280.2	// R_3rd ROT R SERVO RESET
AND NOT   T0815	// -
OUT       D002280.2	// R_3rd ROT R SERVO RESET
TON       T0815 1	// -
; L156
LOAD      F00099
DMOV      D004582 D002288	// R_3rd ROT R A¢Ò¡¾¡¿Au¨ùO
// Currnent Postition
; L158
LOADD=    D004540 D001286
AND       T0515	// -
AND       M01652	// -
OUT       M04150	// -

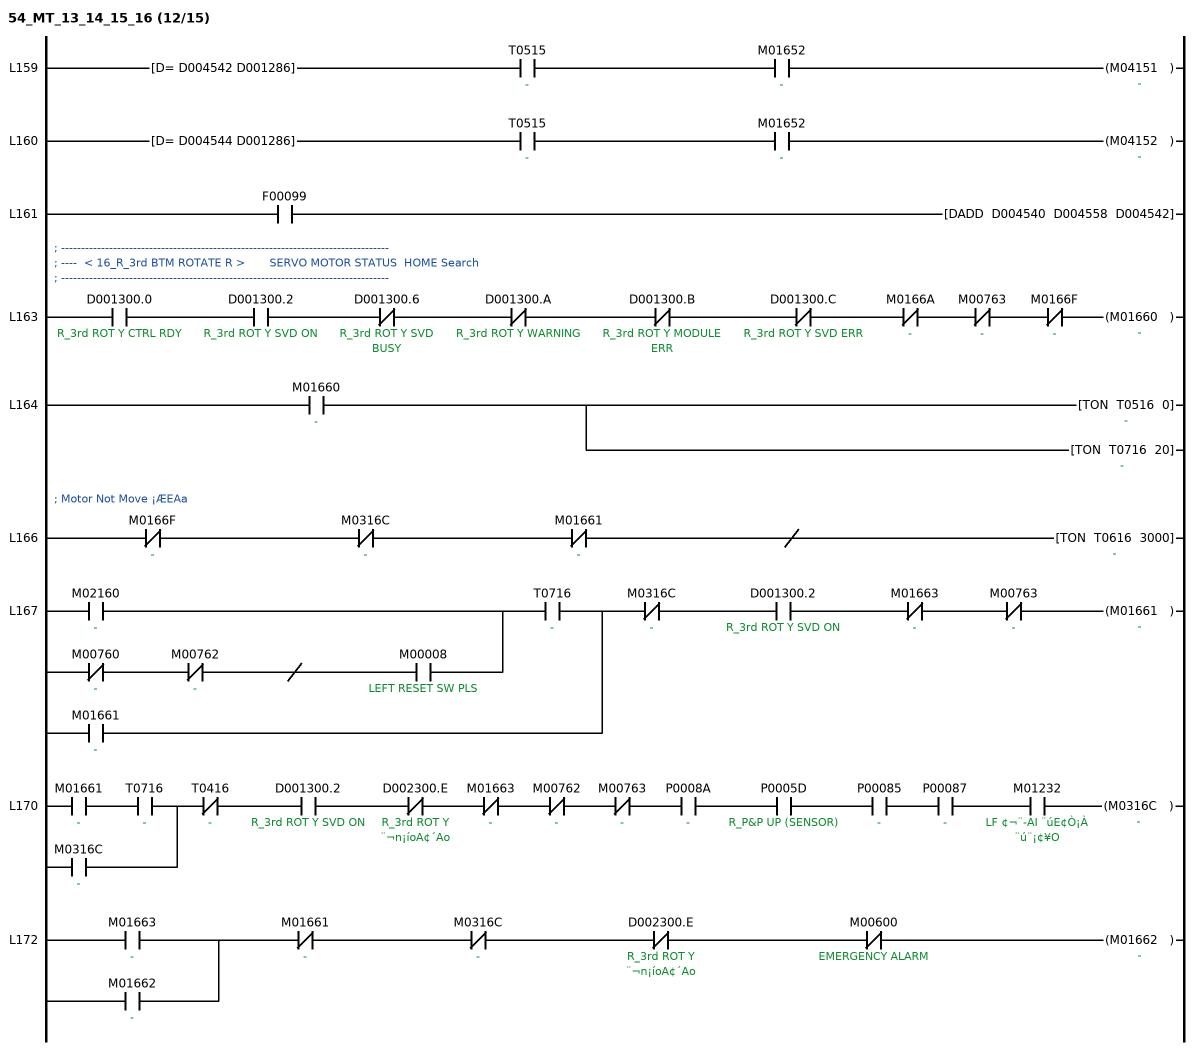
; L159
LOADD=    D004542 D001286
AND       T0515	// -
AND       M01652	// -
OUT       M04151	// -
; L160
LOADD=    D004544 D001286
AND       T0515	// -
AND       M01652	// -
OUT       M04152	// -
; L161
LOAD      F00099
DADD      D004540 D004558 D004542
// ----------------------------------------------------------------------------------
// 
// ----  < 16_R_3rd BTM ROTATE R >       SERVO MOTOR STATUS  HOME Search
// 
// ----------------------------------------------------------------------------------
; L163
LOAD      D001300.0	// R_3rd ROT Y CTRL RDY
AND       D001300.2	// R_3rd ROT Y SVD ON
AND NOT   D001300.6	// R_3rd ROT Y SVD BUSY
AND NOT   D001300.A	// R_3rd ROT Y WARNING
AND NOT   D001300.B	// R_3rd ROT Y MODULE ERR
AND NOT   D001300.C	// R_3rd ROT Y SVD ERR
AND NOT   M0166A	// -
AND NOT   M00763	// -
AND NOT   M0166F	// -
OUT       M01660	// -
; L164
LOAD      M01660	// -
TON       T0516 0	// -
TON       T0716 20	// -
; L166
LOAD NOT  M0166F	// -
AND NOT   M0316C	// -
AND NOT   M01661	// -
NOT
TON       T0616 3000	// -
// output comment: Motor Not Move ¡ÆEAa
; L167
LOAD      M02160	// -
LOAD NOT  M00760	// -
AND NOT   M00762	// -
NOT
AND       M00008	// LEFT RESET SW PLS
OR LOAD
AND       T0716	// -
OR        M01661	// -
AND NOT   M0316C	// -
AND       D001300.2	// R_3rd ROT Y SVD ON
AND NOT   M01663	// -
AND NOT   M00763	// -
OUT       M01661	// -
; L170
LOAD      M01661	// -
AND       T0716	// -
OR        M0316C	// -
AND NOT   T0416	// -
AND       D001300.2	// R_3rd ROT Y SVD ON
AND NOT   D002300.E	// R_3rd ROT Y ¨¬n¡íoA¢´Ao
AND NOT   M01663	// -
AND NOT   M00762	// -
AND NOT   M00763	// -
AND       P0008A	// -
AND       P0005D	// R_P&P UP (SENSOR)
AND       P00085	// -
AND       P00087	// -
AND       M01232	// LF ¢¬¨­AI ¨úE¢Ò¡À ¨ú¨¡¢¥O
OUT       M0316C	// -
; L172
LOAD      M01663	// -
OR        M01662	// -
AND NOT   M01661	// -
AND NOT   M0316C	// -
AND NOT   D002300.E	// R_3rd ROT Y ¨¬n¡íoA¢´Ao
AND NOT   M00600	// EMERGENCY ALARM
OUT       M01662	// -

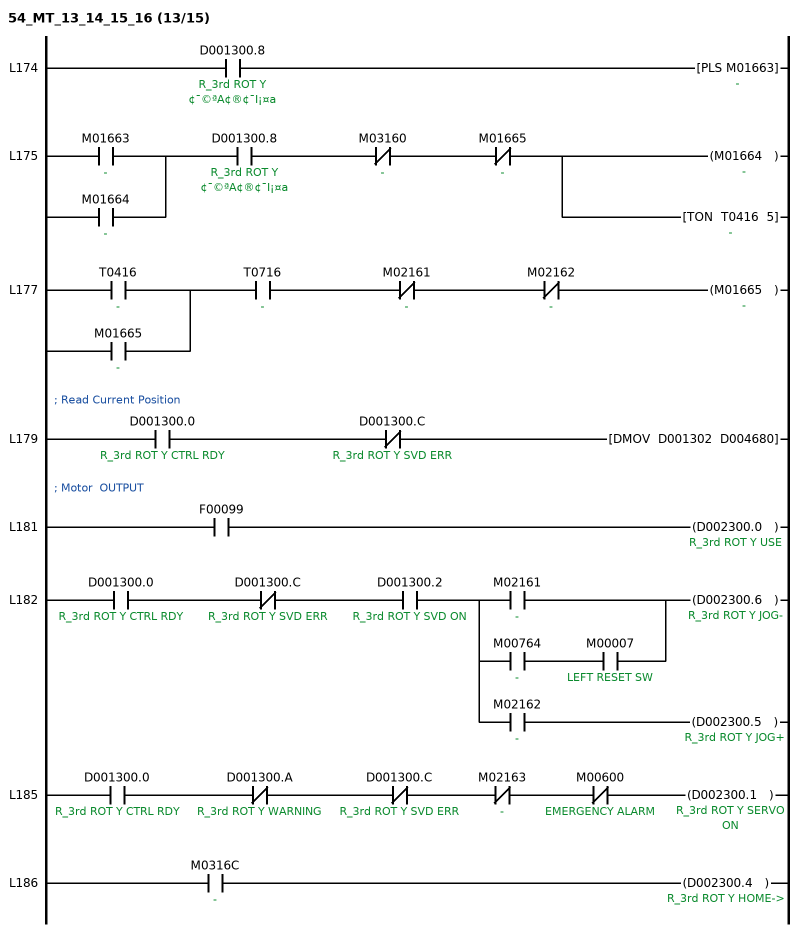
; L174
LOAD      D001300.8	// R_3rd ROT Y ¢¯©ªA¢®¢¯I¡¤a
OUTP      M01663	// -
; L175
LOAD      M01663	// -
OR        M01664	// -
AND       D001300.8	// R_3rd ROT Y ¢¯©ªA¢®¢¯I¡¤a
AND NOT   M03160	// -
AND NOT   M01665	// -
OUT       M01664	// -
TON       T0416 5	// -
; L177
LOAD      T0416	// -
OR        M01665	// -
AND       T0716	// -
AND NOT   M02161	// -
AND NOT   M02162	// -
OUT       M01665	// -
; L179
LOAD      D001300.0	// R_3rd ROT Y CTRL RDY
AND NOT   D001300.C	// R_3rd ROT Y SVD ERR
DMOV      D001302 D004680
// output comment: Read Current Position
//  Motor  OUTPUT
; L181
LOAD      F00099
OUT       D002300.0	// R_3rd ROT Y USE
; L182
LOAD      D001300.0	// R_3rd ROT Y CTRL RDY
AND NOT   D001300.C	// R_3rd ROT Y SVD ERR
AND       D001300.2	// R_3rd ROT Y SVD ON
MPUSH
LOAD      M02161	// -
LOAD      M00764	// -
AND       M00007	// LEFT RESET SW
OR LOAD
AND LOAD
OUT       D002300.6	// R_3rd ROT Y JOG-
MPOP
AND       M02162	// -
OUT       D002300.5	// R_3rd ROT Y JOG+
; L185
LOAD      D001300.0	// R_3rd ROT Y CTRL RDY
AND NOT   D001300.A	// R_3rd ROT Y WARNING
AND NOT   D001300.C	// R_3rd ROT Y SVD ERR
AND NOT   M02163	// -
AND NOT   M00600	// EMERGENCY ALARM
OUT       D002300.1	// R_3rd ROT Y SERVO ON
; L186
LOAD      M0316C	// -
OUT       D002300.4	// R_3rd ROT Y HOME->

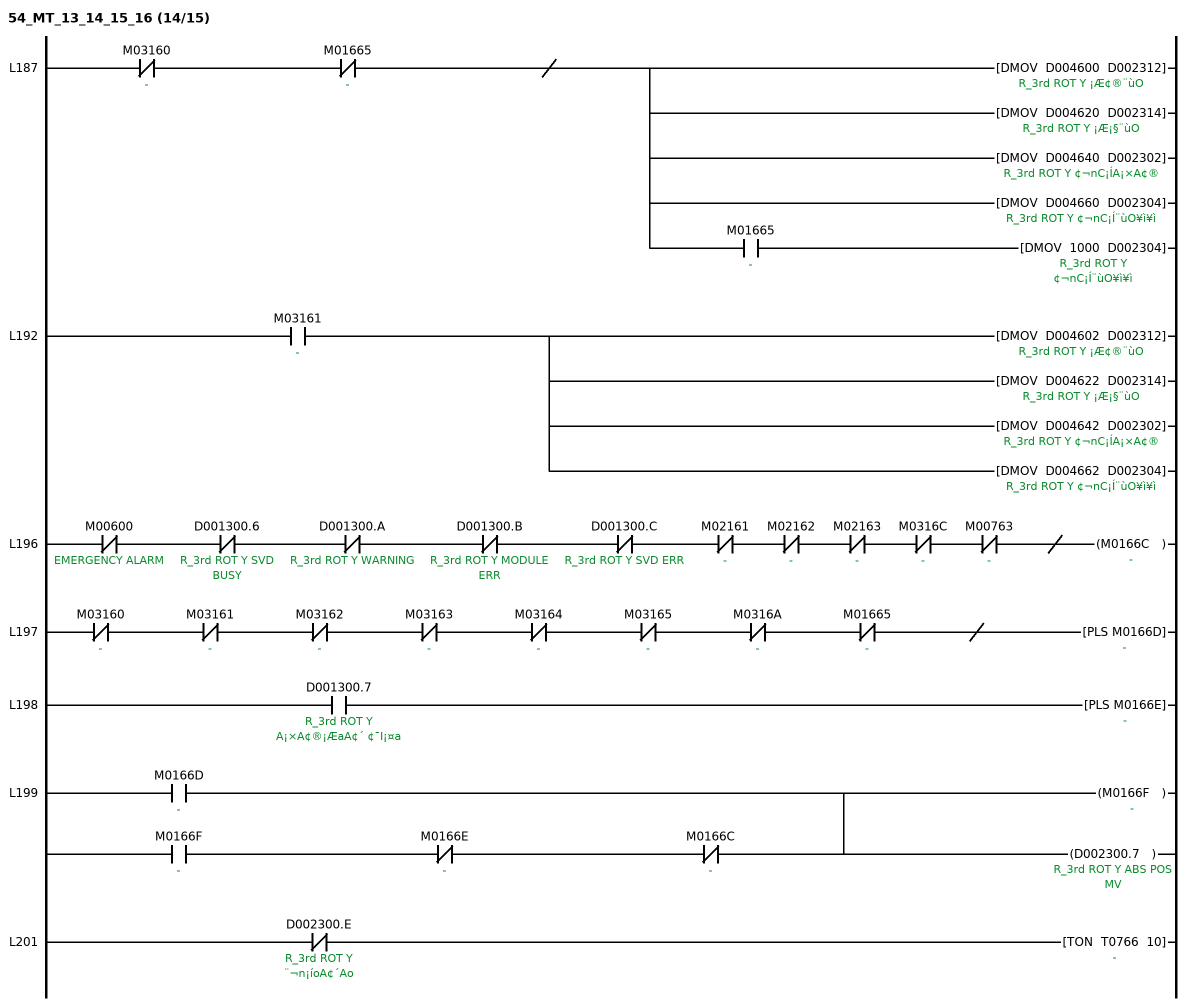
; L187
LOAD NOT  M03160	// -
AND NOT   M01665	// -
NOT
DMOV      D004600 D002312	// R_3rd ROT Y ¡Æ¢®¨ùO
DMOV      D004620 D002314	// R_3rd ROT Y ¡Æ¡§¨ùO
DMOV      D004640 D002302	// R_3rd ROT Y ¢¬nC¡ÍA¡×A¢®
DMOV      D004660 D002304	// R_3rd ROT Y ¢¬nC¡Í¨ùO¥ì¥ì
AND       M01665	// -
DMOV      1000 D002304	// R_3rd ROT Y ¢¬nC¡Í¨ùO¥ì¥ì
; L192
LOAD      M03161	// -
DMOV      D004602 D002312	// R_3rd ROT Y ¡Æ¢®¨ùO
DMOV      D004622 D002314	// R_3rd ROT Y ¡Æ¡§¨ùO
DMOV      D004642 D002302	// R_3rd ROT Y ¢¬nC¡ÍA¡×A¢®
DMOV      D004662 D002304	// R_3rd ROT Y ¢¬nC¡Í¨ùO¥ì¥ì
; L196
LOAD NOT  M00600	// EMERGENCY ALARM
AND NOT   D001300.6	// R_3rd ROT Y SVD BUSY
AND NOT   D001300.A	// R_3rd ROT Y WARNING
AND NOT   D001300.B	// R_3rd ROT Y MODULE ERR
AND NOT   D001300.C	// R_3rd ROT Y SVD ERR
AND NOT   M02161	// -
AND NOT   M02162	// -
AND NOT   M02163	// -
AND NOT   M0316C	// -
AND NOT   M00763	// -
NOT
OUT       M0166C	// -
; L197
LOAD NOT  M03160	// -
AND NOT   M03161	// -
AND NOT   M03162	// -
AND NOT   M03163	// -
AND NOT   M03164	// -
AND NOT   M03165	// -
AND NOT   M0316A	// -
AND NOT   M01665	// -
NOT
OUTP      M0166D	// -
; L198
LOAD      D001300.7	// R_3rd ROT Y A¡×A¢®¡ÆaA¢´ ¢¯I¡¤a
OUTP      M0166E	// -
; L199
LOAD      M0166D	// -
LOAD      M0166F	// -
AND NOT   M0166E	// -
AND NOT   M0166C	// -
OR LOAD
OUT       M0166F	// -
OUT       D002300.7	// R_3rd ROT Y ABS POS MV
; L201
LOAD NOT  D002300.E	// R_3rd ROT Y ¨¬n¡íoA¢´Ao
TON       T0766 10	// -

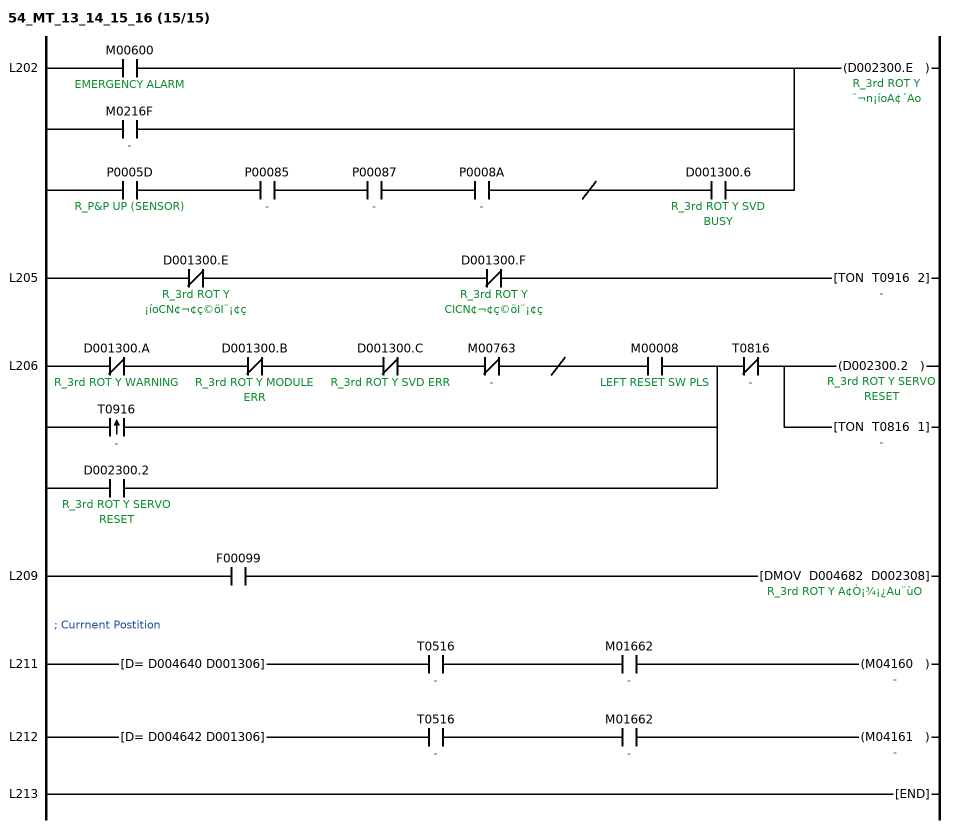
; L202
LOAD      M00600	// EMERGENCY ALARM
OR        M0216F	// -
LOAD      P0005D	// R_P&P UP (SENSOR)
AND       P00085	// -
AND       P00087	// -
AND       P0008A	// -
NOT
AND       D001300.6	// R_3rd ROT Y SVD BUSY
OR LOAD
OUT       D002300.E	// R_3rd ROT Y ¨¬n¡íoA¢´Ao
; L205
LOAD NOT  D001300.E	// R_3rd ROT Y ¡íoCN¢¬¢ç©öI¨¡¢ç
AND NOT   D001300.F	// R_3rd ROT Y CICN¢¬¢ç©öI¨¡¢ç
TON       T0916 2	// -
; L206
LOAD NOT  D001300.A	// R_3rd ROT Y WARNING
AND NOT   D001300.B	// R_3rd ROT Y MODULE ERR
AND NOT   D001300.C	// R_3rd ROT Y SVD ERR
AND NOT   M00763	// -
NOT
AND       M00008	// LEFT RESET SW PLS
ORP       T0916	// -
OR        D002300.2	// R_3rd ROT Y SERVO RESET
AND NOT   T0816	// -
OUT       D002300.2	// R_3rd ROT Y SERVO RESET
TON       T0816 1	// -
; L209
LOAD      F00099
DMOV      D004682 D002308	// R_3rd ROT Y A¢Ò¡¾¡¿Au¨ùO
// Currnent Postition
; L211
LOADD=    D004640 D001306
AND       T0516	// -
AND       M01662	// -
OUT       M04160	// -
; L212
LOADD=    D004642 D001306
AND       T0516	// -
AND       M01662	// -
OUT       M04161	// -
; L213
END

PROGRAM 55_MT_17_18_19_20 (task: ¨ö¨¬A¥ì CA¡¤I¡¾¡¿¡¤¡Í)

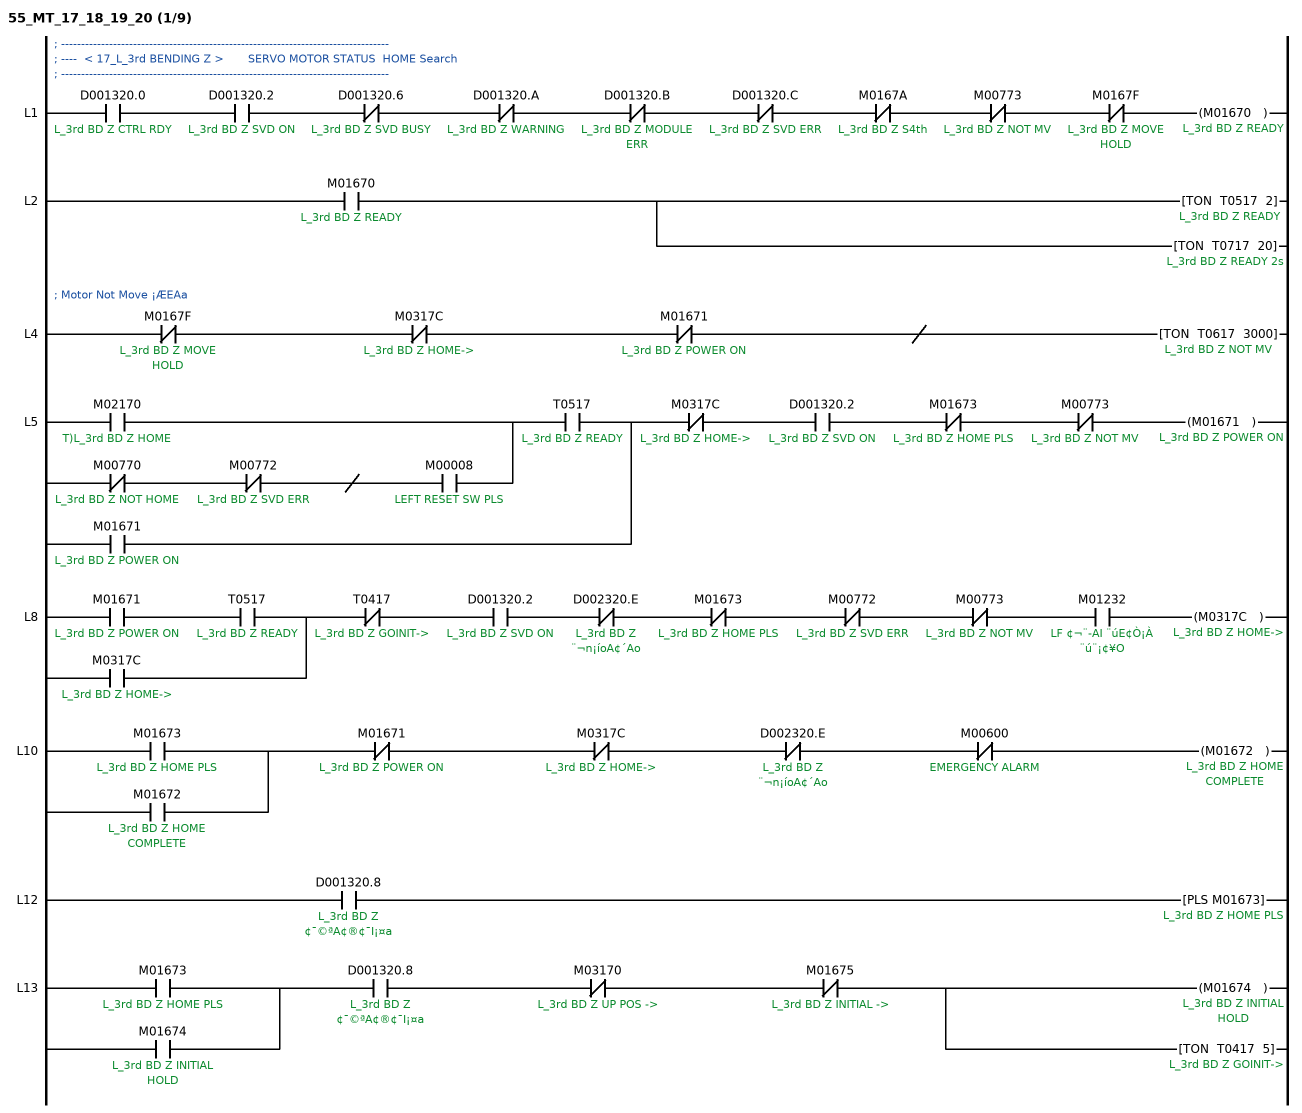
// ----------------------------------------------------------------------------------
// 
// ----  < 17_L_3rd BENDING Z >       SERVO MOTOR STATUS  HOME Search
// 
// ----------------------------------------------------------------------------------
; L1
LOAD      D001320.0	// L_3rd BD Z CTRL RDY
AND       D001320.2	// L_3rd BD Z SVD ON
AND NOT   D001320.6	// L_3rd BD Z SVD BUSY
AND NOT   D001320.A	// L_3rd BD Z WARNING
AND NOT   D001320.B	// L_3rd BD Z MODULE ERR
AND NOT   D001320.C	// L_3rd BD Z SVD ERR
AND NOT   M0167A	// L_3rd BD Z S4th
AND NOT   M00773	// L_3rd BD Z NOT MV
AND NOT   M0167F	// L_3rd BD Z MOVE HOLD
OUT       M01670	// L_3rd BD Z READY
; L2
LOAD      M01670	// L_3rd BD Z READY
TON       T0517 2	// L_3rd BD Z READY
TON       T0717 20	// L_3rd BD Z READY 2s
; L4
LOAD NOT  M0167F	// L_3rd BD Z MOVE HOLD
AND NOT   M0317C	// L_3rd BD Z HOME->
AND NOT   M01671	// L_3rd BD Z POWER ON
NOT
TON       T0617 3000	// L_3rd BD Z NOT MV
// output comment: Motor Not Move ¡ÆEAa
; L5
LOAD      M02170	// T)L_3rd BD Z HOME
LOAD NOT  M00770	// L_3rd BD Z NOT HOME
AND NOT   M00772	// L_3rd BD Z SVD ERR
NOT
AND       M00008	// LEFT RESET SW PLS
OR LOAD
AND       T0517	// L_3rd BD Z READY
OR        M01671	// L_3rd BD Z POWER ON
AND NOT   M0317C	// L_3rd BD Z HOME->
AND       D001320.2	// L_3rd BD Z SVD ON
AND NOT   M01673	// L_3rd BD Z HOME PLS
AND NOT   M00773	// L_3rd BD Z NOT MV
OUT       M01671	// L_3rd BD Z POWER ON
; L8
LOAD      M01671	// L_3rd BD Z POWER ON
AND       T0517	// L_3rd BD Z READY
OR        M0317C	// L_3rd BD Z HOME->
AND NOT   T0417	// L_3rd BD Z GOINIT->
AND       D001320.2	// L_3rd BD Z SVD ON
AND NOT   D002320.E	// L_3rd BD Z ¨¬n¡íoA¢´Ao
AND NOT   M01673	// L_3rd BD Z HOME PLS
AND NOT   M00772	// L_3rd BD Z SVD ERR
AND NOT   M00773	// L_3rd BD Z NOT MV
AND       M01232	// LF ¢¬¨­AI ¨úE¢Ò¡À ¨ú¨¡¢¥O
OUT       M0317C	// L_3rd BD Z HOME->
; L10
LOAD      M01673	// L_3rd BD Z HOME PLS
OR        M01672	// L_3rd BD Z HOME COMPLETE
AND NOT   M01671	// L_3rd BD Z POWER ON
AND NOT   M0317C	// L_3rd BD Z HOME->
AND NOT   D002320.E	// L_3rd BD Z ¨¬n¡íoA¢´Ao
AND NOT   M00600	// EMERGENCY ALARM
OUT       M01672	// L_3rd BD Z HOME COMPLETE
; L12
LOAD      D001320.8	// L_3rd BD Z ¢¯©ªA¢®¢¯I¡¤a
OUTP      M01673	// L_3rd BD Z HOME PLS
; L13
LOAD      M01673	// L_3rd BD Z HOME PLS
OR        M01674	// L_3rd BD Z INITIAL HOLD
AND       D001320.8	// L_3rd BD Z ¢¯©ªA¢®¢¯I¡¤a
AND NOT   M03170	// L_3rd BD Z UP POS ->
AND NOT   M01675	// L_3rd BD Z INITIAL ->
OUT       M01674	// L_3rd BD Z INITIAL HOLD
TON       T0417 5	// L_3rd BD Z GOINIT->

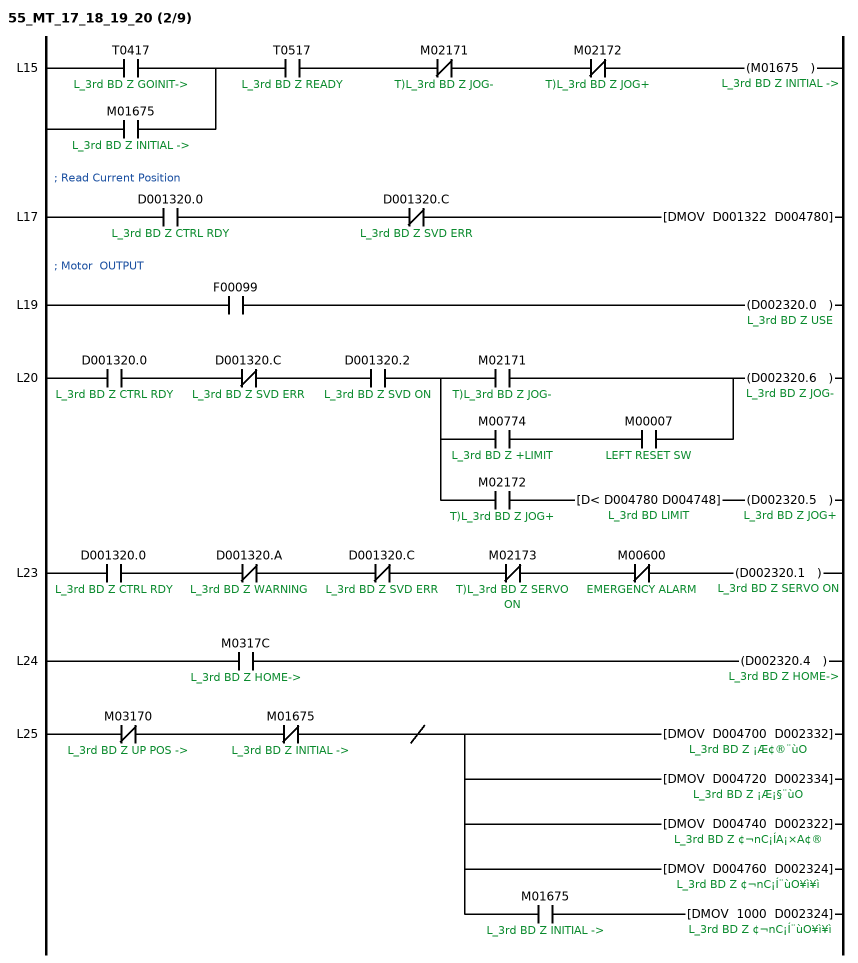
; L15
LOAD      T0417	// L_3rd BD Z GOINIT->
OR        M01675	// L_3rd BD Z INITIAL ->
AND       T0517	// L_3rd BD Z READY
AND NOT   M02171	// T)L_3rd BD Z JOG-
AND NOT   M02172	// T)L_3rd BD Z JOG+
OUT       M01675	// L_3rd BD Z INITIAL ->
; L17
LOAD      D001320.0	// L_3rd BD Z CTRL RDY
AND NOT   D001320.C	// L_3rd BD Z SVD ERR
DMOV      D001322 D004780
// output comment: Read Current Position
//  Motor  OUTPUT
; L19
LOAD      F00099
OUT       D002320.0	// L_3rd BD Z USE
; L20
LOAD      D001320.0	// L_3rd BD Z CTRL RDY
AND NOT   D001320.C	// L_3rd BD Z SVD ERR
AND       D001320.2	// L_3rd BD Z SVD ON
MPUSH
LOAD      M02171	// T)L_3rd BD Z JOG-
LOAD      M00774	// L_3rd BD Z +LIMIT
AND       M00007	// LEFT RESET SW
OR LOAD
AND LOAD
OUT       D002320.6	// L_3rd BD Z JOG-
MPOP
AND       M02172	// T)L_3rd BD Z JOG+
ANDD<     D004780 D004748	// L_3rd BD LIMIT
OUT       D002320.5	// L_3rd BD Z JOG+
; L23
LOAD      D001320.0	// L_3rd BD Z CTRL RDY
AND NOT   D001320.A	// L_3rd BD Z WARNING
AND NOT   D001320.C	// L_3rd BD Z SVD ERR
AND NOT   M02173	// T)L_3rd BD Z SERVO ON
AND NOT   M00600	// EMERGENCY ALARM
OUT       D002320.1	// L_3rd BD Z SERVO ON
; L24
LOAD      M0317C	// L_3rd BD Z HOME->
OUT       D002320.4	// L_3rd BD Z HOME->
; L25
LOAD NOT  M03170	// L_3rd BD Z UP POS ->
AND NOT   M01675	// L_3rd BD Z INITIAL ->
NOT
DMOV      D004700 D002332	// L_3rd BD Z ¡Æ¢®¨ùO
DMOV      D004720 D002334	// L_3rd BD Z ¡Æ¡§¨ùO
DMOV      D004740 D002322	// L_3rd BD Z ¢¬nC¡ÍA¡×A¢®
DMOV      D004760 D002324	// L_3rd BD Z ¢¬nC¡Í¨ùO¥ì¥ì
AND       M01675	// L_3rd BD Z INITIAL ->
DMOV      1000 D002324	// L_3rd BD Z ¢¬nC¡Í¨ùO¥ì¥ì

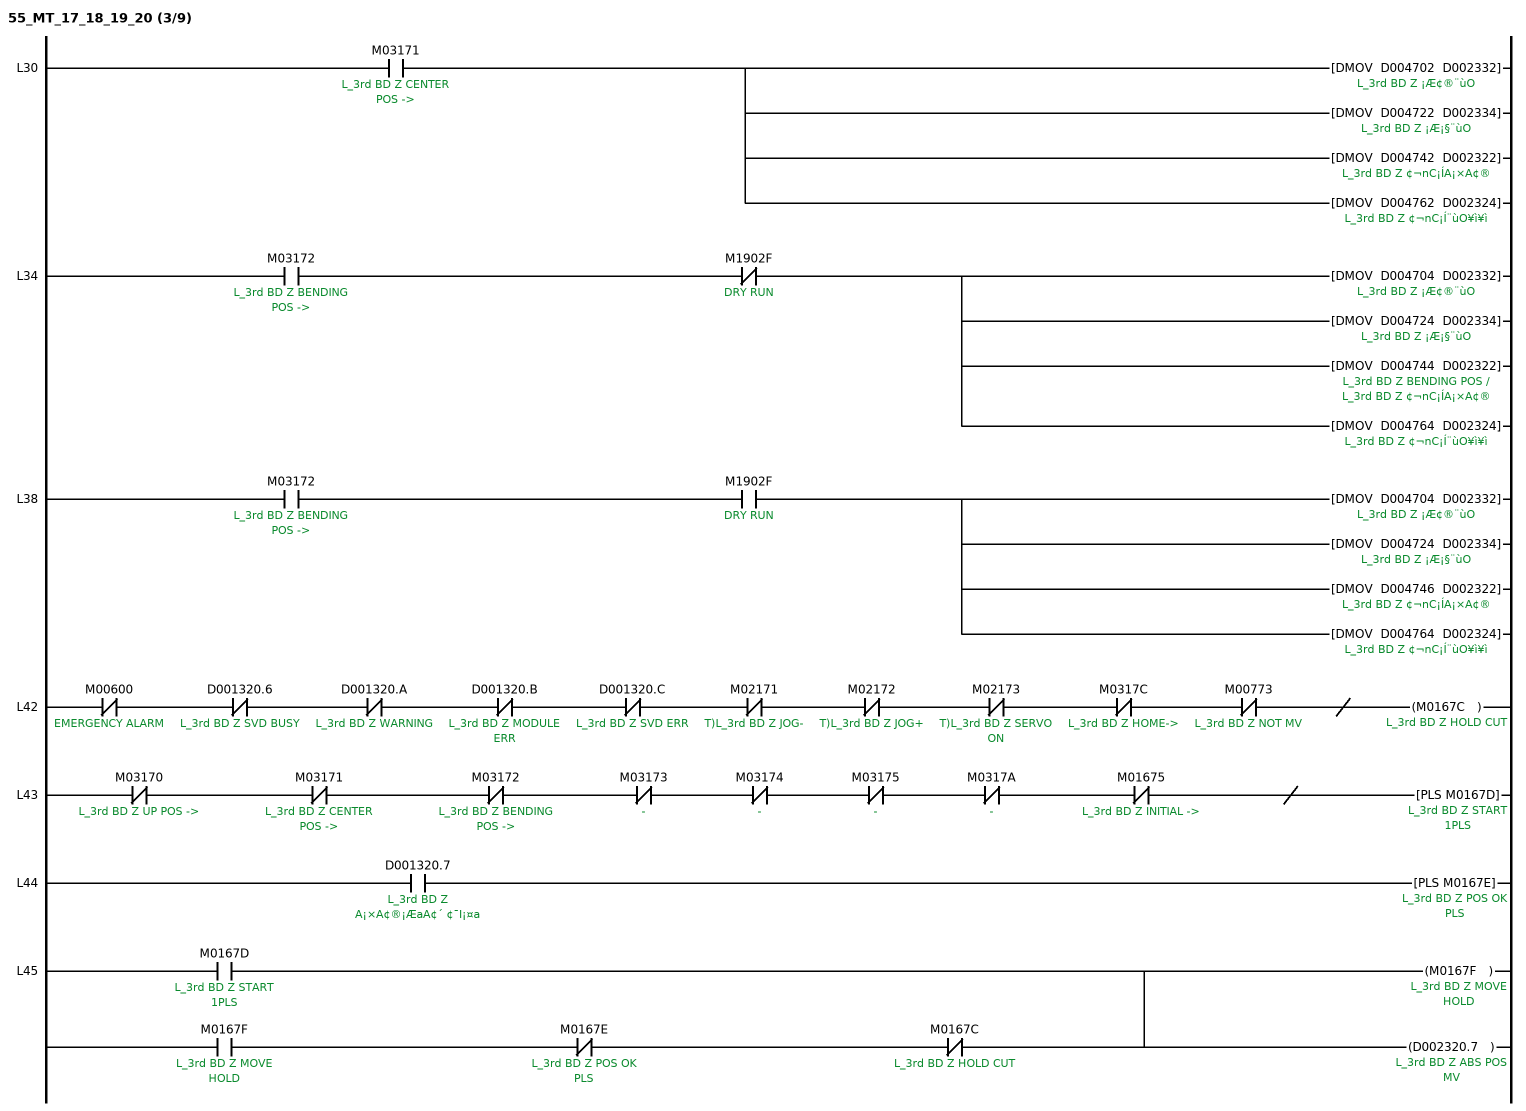
; L30
LOAD      M03171	// L_3rd BD Z CENTER POS ->
DMOV      D004702 D002332	// L_3rd BD Z ¡Æ¢®¨ùO
DMOV      D004722 D002334	// L_3rd BD Z ¡Æ¡§¨ùO
DMOV      D004742 D002322	// L_3rd BD Z ¢¬nC¡ÍA¡×A¢®
DMOV      D004762 D002324	// L_3rd BD Z ¢¬nC¡Í¨ùO¥ì¥ì
; L34
LOAD      M03172	// L_3rd BD Z BENDING POS ->
AND NOT   M1902F	// DRY RUN
DMOV      D004704 D002332	// L_3rd BD Z ¡Æ¢®¨ùO
DMOV      D004724 D002334	// L_3rd BD Z ¡Æ¡§¨ùO
DMOV      D004744 D002322	// L_3rd BD Z BENDING POS / L_3rd BD Z ¢¬nC¡ÍA¡×A¢®
DMOV      D004764 D002324	// L_3rd BD Z ¢¬nC¡Í¨ùO¥ì¥ì
; L38
LOAD      M03172	// L_3rd BD Z BENDING POS ->
AND       M1902F	// DRY RUN
DMOV      D004704 D002332	// L_3rd BD Z ¡Æ¢®¨ùO
DMOV      D004724 D002334	// L_3rd BD Z ¡Æ¡§¨ùO
DMOV      D004746 D002322	// L_3rd BD Z ¢¬nC¡ÍA¡×A¢®
DMOV      D004764 D002324	// L_3rd BD Z ¢¬nC¡Í¨ùO¥ì¥ì
; L42
LOAD NOT  M00600	// EMERGENCY ALARM
AND NOT   D001320.6	// L_3rd BD Z SVD BUSY
AND NOT   D001320.A	// L_3rd BD Z WARNING
AND NOT   D001320.B	// L_3rd BD Z MODULE ERR
AND NOT   D001320.C	// L_3rd BD Z SVD ERR
AND NOT   M02171	// T)L_3rd BD Z JOG-
AND NOT   M02172	// T)L_3rd BD Z JOG+
AND NOT   M02173	// T)L_3rd BD Z SERVO ON
AND NOT   M0317C	// L_3rd BD Z HOME->
AND NOT   M00773	// L_3rd BD Z NOT MV
NOT
OUT       M0167C	// L_3rd BD Z HOLD CUT
; L43
LOAD NOT  M03170	// L_3rd BD Z UP POS ->
AND NOT   M03171	// L_3rd BD Z CENTER POS ->
AND NOT   M03172	// L_3rd BD Z BENDING POS ->
AND NOT   M03173	// -
AND NOT   M03174	// -
AND NOT   M03175	// -
AND NOT   M0317A	// -
AND NOT   M01675	// L_3rd BD Z INITIAL ->
NOT
OUTP      M0167D	// L_3rd BD Z START 1PLS
; L44
LOAD      D001320.7	// L_3rd BD Z A¡×A¢®¡ÆaA¢´ ¢¯I¡¤a
OUTP      M0167E	// L_3rd BD Z POS OK PLS
; L45
LOAD      M0167D	// L_3rd BD Z START 1PLS
LOAD      M0167F	// L_3rd BD Z MOVE HOLD
AND NOT   M0167E	// L_3rd BD Z POS OK PLS
AND NOT   M0167C	// L_3rd BD Z HOLD CUT
OR LOAD
OUT       M0167F	// L_3rd BD Z MOVE HOLD
OUT       D002320.7	// L_3rd BD Z ABS POS MV

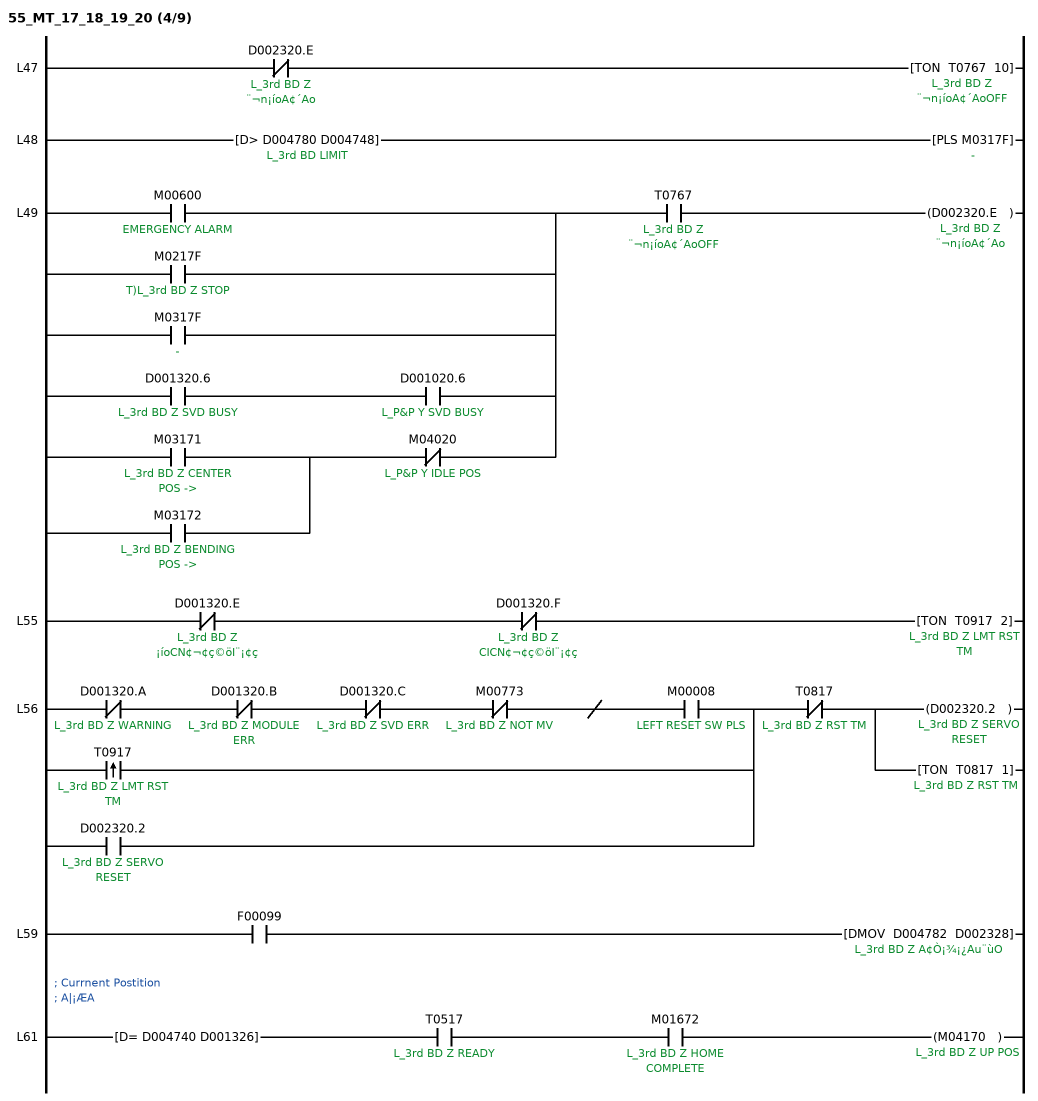
; L47
LOAD NOT  D002320.E	// L_3rd BD Z ¨¬n¡íoA¢´Ao
TON       T0767 10	// L_3rd BD Z ¨¬n¡íoA¢´AoOFF
; L48
LOADD>    D004780 D004748	// L_3rd BD LIMIT
OUTP      M0317F	// -
; L49
LOAD      M00600	// EMERGENCY ALARM
OR        M0217F	// T)L_3rd BD Z STOP
OR        M0317F	// -
LOAD      D001320.6	// L_3rd BD Z SVD BUSY
AND       D001020.6	// L_P&P Y SVD BUSY
OR LOAD
LOAD      M03171	// L_3rd BD Z CENTER POS ->
OR        M03172	// L_3rd BD Z BENDING POS ->
AND NOT   M04020	// L_P&P Y IDLE POS
OR LOAD
AND       T0767	// L_3rd BD Z ¨¬n¡íoA¢´AoOFF
OUT       D002320.E	// L_3rd BD Z ¨¬n¡íoA¢´Ao
; L55
LOAD NOT  D001320.E	// L_3rd BD Z ¡íoCN¢¬¢ç©öI¨¡¢ç
AND NOT   D001320.F	// L_3rd BD Z CICN¢¬¢ç©öI¨¡¢ç
TON       T0917 2	// L_3rd BD Z LMT RST TM
; L56
LOAD NOT  D001320.A	// L_3rd BD Z WARNING
AND NOT   D001320.B	// L_3rd BD Z MODULE ERR
AND NOT   D001320.C	// L_3rd BD Z SVD ERR
AND NOT   M00773	// L_3rd BD Z NOT MV
NOT
AND       M00008	// LEFT RESET SW PLS
ORP       T0917	// L_3rd BD Z LMT RST TM
OR        D002320.2	// L_3rd BD Z SERVO RESET
AND NOT   T0817	// L_3rd BD Z RST TM
OUT       D002320.2	// L_3rd BD Z SERVO RESET
TON       T0817 1	// L_3rd BD Z RST TM
; L59
LOAD      F00099
DMOV      D004782 D002328	// L_3rd BD Z A¢Ò¡¾¡¿Au¨ùO
// Currnent Postition
; L61
LOADD=    D004740 D001326
AND       T0517	// L_3rd BD Z READY
AND       M01672	// L_3rd BD Z HOME COMPLETE
OUT       M04170	// L_3rd BD Z UP POS
// output comment: A|¡ÆA

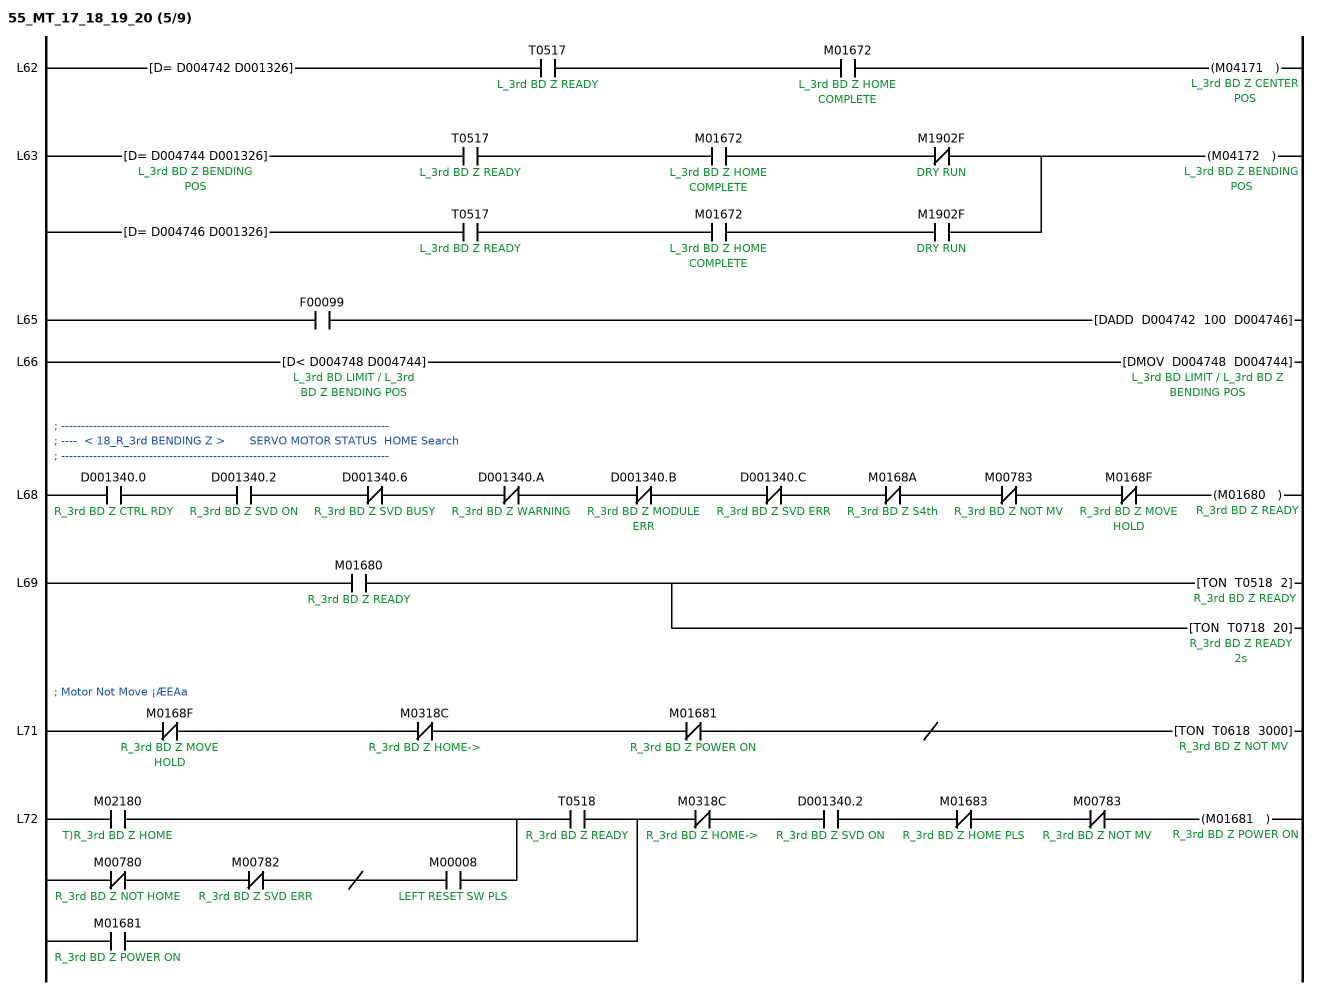
; L62
LOADD=    D004742 D001326
AND       T0517	// L_3rd BD Z READY
AND       M01672	// L_3rd BD Z HOME COMPLETE
OUT       M04171	// L_3rd BD Z CENTER POS
; L63
LOADD=    D004744 D001326	// L_3rd BD Z BENDING POS
AND       T0517	// L_3rd BD Z READY
AND       M01672	// L_3rd BD Z HOME COMPLETE
AND NOT   M1902F	// DRY RUN
LOADD=    D004746 D001326
AND       T0517	// L_3rd BD Z READY
AND       M01672	// L_3rd BD Z HOME COMPLETE
AND       M1902F	// DRY RUN
OR LOAD
OUT       M04172	// L_3rd BD Z BENDING POS
; L65
LOAD      F00099
DADD      D004742 100 D004746
; L66
LOADD<    D004748 D004744	// L_3rd BD LIMIT / L_3rd BD Z BENDING POS
DMOV      D004748 D004744	// L_3rd BD LIMIT / L_3rd BD Z BENDING POS
// ----------------------------------------------------------------------------------
// 
// ----  < 18_R_3rd BENDING Z >       SERVO MOTOR STATUS  HOME Search
// 
// ----------------------------------------------------------------------------------
; L68
LOAD      D001340.0	// R_3rd BD Z CTRL RDY
AND       D001340.2	// R_3rd BD Z SVD ON
AND NOT   D001340.6	// R_3rd BD Z SVD BUSY
AND NOT   D001340.A	// R_3rd BD Z WARNING
AND NOT   D001340.B	// R_3rd BD Z MODULE ERR
AND NOT   D001340.C	// R_3rd BD Z SVD ERR
AND NOT   M0168A	// R_3rd BD Z S4th
AND NOT   M00783	// R_3rd BD Z NOT MV
AND NOT   M0168F	// R_3rd BD Z MOVE HOLD
OUT       M01680	// R_3rd BD Z READY
; L69
LOAD      M01680	// R_3rd BD Z READY
TON       T0518 2	// R_3rd BD Z READY
TON       T0718 20	// R_3rd BD Z READY 2s
; L71
LOAD NOT  M0168F	// R_3rd BD Z MOVE HOLD
AND NOT   M0318C	// R_3rd BD Z HOME->
AND NOT   M01681	// R_3rd BD Z POWER ON
NOT
TON       T0618 3000	// R_3rd BD Z NOT MV
// output comment: Motor Not Move ¡ÆEAa
; L72
LOAD      M02180	// T)R_3rd BD Z HOME
LOAD NOT  M00780	// R_3rd BD Z NOT HOME
AND NOT   M00782	// R_3rd BD Z SVD ERR
NOT
AND       M00008	// LEFT RESET SW PLS
OR LOAD
AND       T0518	// R_3rd BD Z READY
OR        M01681	// R_3rd BD Z POWER ON
AND NOT   M0318C	// R_3rd BD Z HOME->
AND       D001340.2	// R_3rd BD Z SVD ON
AND NOT   M01683	// R_3rd BD Z HOME PLS
AND NOT   M00783	// R_3rd BD Z NOT MV
OUT       M01681	// R_3rd BD Z POWER ON

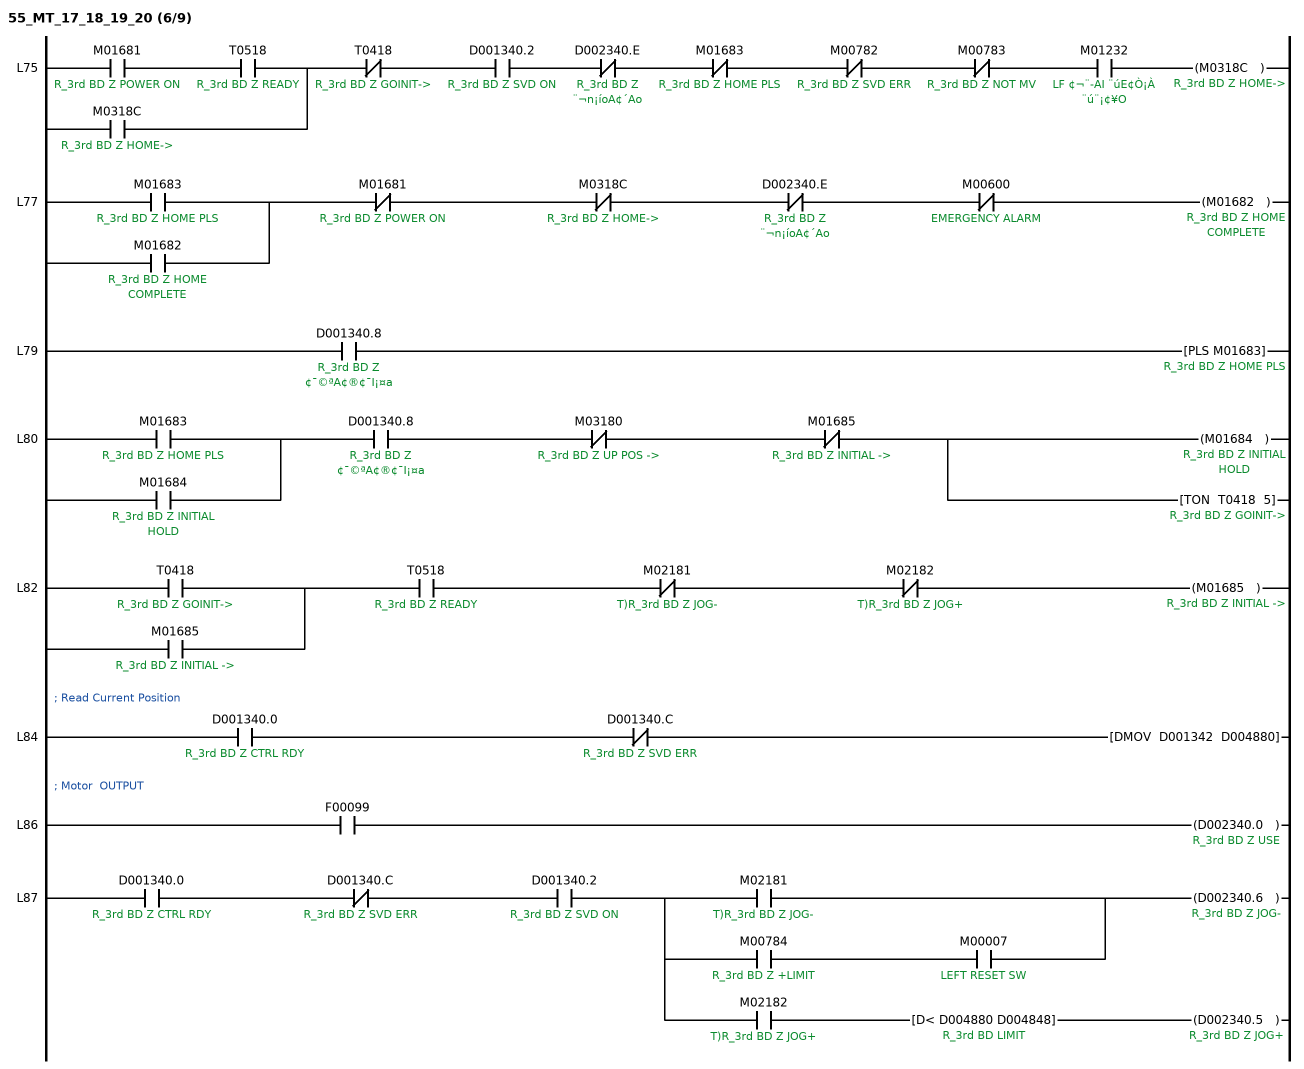
; L75
LOAD      M01681	// R_3rd BD Z POWER ON
AND       T0518	// R_3rd BD Z READY
OR        M0318C	// R_3rd BD Z HOME->
AND NOT   T0418	// R_3rd BD Z GOINIT->
AND       D001340.2	// R_3rd BD Z SVD ON
AND NOT   D002340.E	// R_3rd BD Z ¨¬n¡íoA¢´Ao
AND NOT   M01683	// R_3rd BD Z HOME PLS
AND NOT   M00782	// R_3rd BD Z SVD ERR
AND NOT   M00783	// R_3rd BD Z NOT MV
AND       M01232	// LF ¢¬¨­AI ¨úE¢Ò¡À ¨ú¨¡¢¥O
OUT       M0318C	// R_3rd BD Z HOME->
; L77
LOAD      M01683	// R_3rd BD Z HOME PLS
OR        M01682	// R_3rd BD Z HOME COMPLETE
AND NOT   M01681	// R_3rd BD Z POWER ON
AND NOT   M0318C	// R_3rd BD Z HOME->
AND NOT   D002340.E	// R_3rd BD Z ¨¬n¡íoA¢´Ao
AND NOT   M00600	// EMERGENCY ALARM
OUT       M01682	// R_3rd BD Z HOME COMPLETE
; L79
LOAD      D001340.8	// R_3rd BD Z ¢¯©ªA¢®¢¯I¡¤a
OUTP      M01683	// R_3rd BD Z HOME PLS
; L80
LOAD      M01683	// R_3rd BD Z HOME PLS
OR        M01684	// R_3rd BD Z INITIAL HOLD
AND       D001340.8	// R_3rd BD Z ¢¯©ªA¢®¢¯I¡¤a
AND NOT   M03180	// R_3rd BD Z UP POS ->
AND NOT   M01685	// R_3rd BD Z INITIAL ->
OUT       M01684	// R_3rd BD Z INITIAL HOLD
TON       T0418 5	// R_3rd BD Z GOINIT->
; L82
LOAD      T0418	// R_3rd BD Z GOINIT->
OR        M01685	// R_3rd BD Z INITIAL ->
AND       T0518	// R_3rd BD Z READY
AND NOT   M02181	// T)R_3rd BD Z JOG-
AND NOT   M02182	// T)R_3rd BD Z JOG+
OUT       M01685	// R_3rd BD Z INITIAL ->
; L84
LOAD      D001340.0	// R_3rd BD Z CTRL RDY
AND NOT   D001340.C	// R_3rd BD Z SVD ERR
DMOV      D001342 D004880
// output comment: Read Current Position
//  Motor  OUTPUT
; L86
LOAD      F00099
OUT       D002340.0	// R_3rd BD Z USE
; L87
LOAD      D001340.0	// R_3rd BD Z CTRL RDY
AND NOT   D001340.C	// R_3rd BD Z SVD ERR
AND       D001340.2	// R_3rd BD Z SVD ON
MPUSH
LOAD      M02181	// T)R_3rd BD Z JOG-
LOAD      M00784	// R_3rd BD Z +LIMIT
AND       M00007	// LEFT RESET SW
OR LOAD
AND LOAD
OUT       D002340.6	// R_3rd BD Z JOG-
MPOP
AND       M02182	// T)R_3rd BD Z JOG+
ANDD<     D004880 D004848	// R_3rd BD LIMIT
OUT       D002340.5	// R_3rd BD Z JOG+

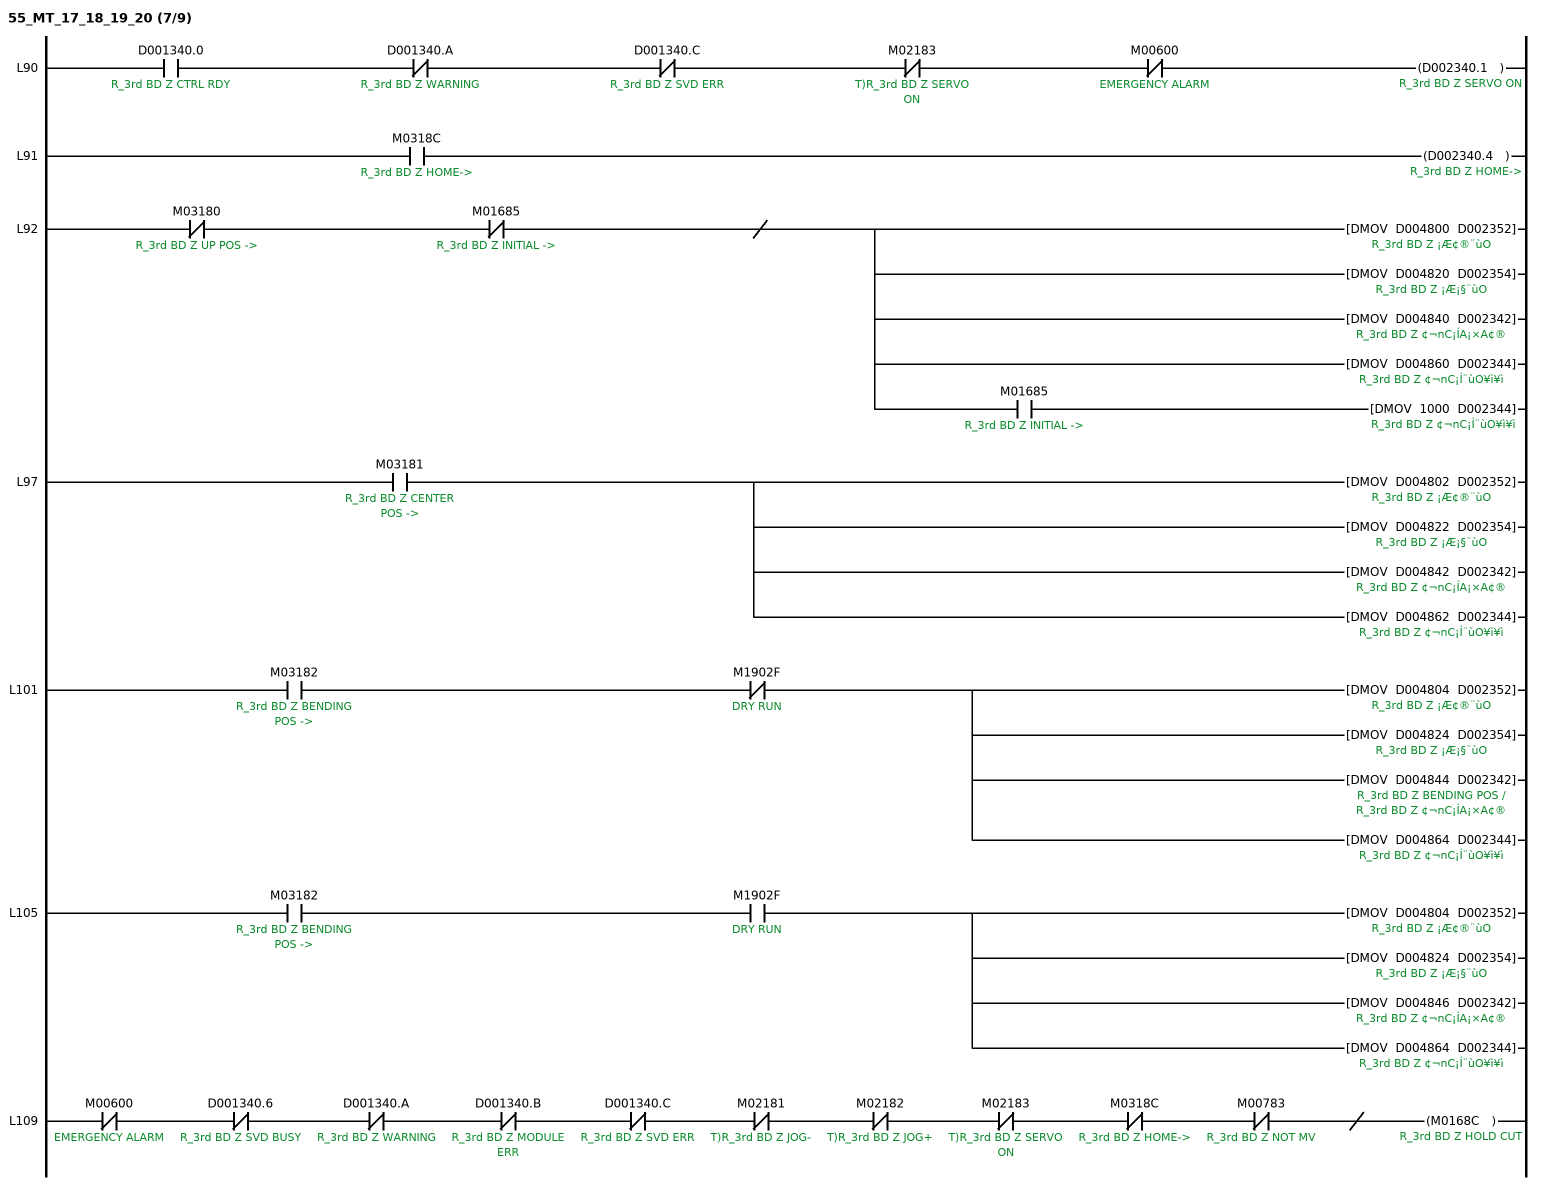
; L90
LOAD      D001340.0	// R_3rd BD Z CTRL RDY
AND NOT   D001340.A	// R_3rd BD Z WARNING
AND NOT   D001340.C	// R_3rd BD Z SVD ERR
AND NOT   M02183	// T)R_3rd BD Z SERVO ON
AND NOT   M00600	// EMERGENCY ALARM
OUT       D002340.1	// R_3rd BD Z SERVO ON
; L91
LOAD      M0318C	// R_3rd BD Z HOME->
OUT       D002340.4	// R_3rd BD Z HOME->
; L92
LOAD NOT  M03180	// R_3rd BD Z UP POS ->
AND NOT   M01685	// R_3rd BD Z INITIAL ->
NOT
DMOV      D004800 D002352	// R_3rd BD Z ¡Æ¢®¨ùO
DMOV      D004820 D002354	// R_3rd BD Z ¡Æ¡§¨ùO
DMOV      D004840 D002342	// R_3rd BD Z ¢¬nC¡ÍA¡×A¢®
DMOV      D004860 D002344	// R_3rd BD Z ¢¬nC¡Í¨ùO¥ì¥ì
AND       M01685	// R_3rd BD Z INITIAL ->
DMOV      1000 D002344	// R_3rd BD Z ¢¬nC¡Í¨ùO¥ì¥ì
; L97
LOAD      M03181	// R_3rd BD Z CENTER POS ->
DMOV      D004802 D002352	// R_3rd BD Z ¡Æ¢®¨ùO
DMOV      D004822 D002354	// R_3rd BD Z ¡Æ¡§¨ùO
DMOV      D004842 D002342	// R_3rd BD Z ¢¬nC¡ÍA¡×A¢®
DMOV      D004862 D002344	// R_3rd BD Z ¢¬nC¡Í¨ùO¥ì¥ì
; L101
LOAD      M03182	// R_3rd BD Z BENDING POS ->
AND NOT   M1902F	// DRY RUN
DMOV      D004804 D002352	// R_3rd BD Z ¡Æ¢®¨ùO
DMOV      D004824 D002354	// R_3rd BD Z ¡Æ¡§¨ùO
DMOV      D004844 D002342	// R_3rd BD Z BENDING POS / R_3rd BD Z ¢¬nC¡ÍA¡×A¢®
DMOV      D004864 D002344	// R_3rd BD Z ¢¬nC¡Í¨ùO¥ì¥ì
; L105
LOAD      M03182	// R_3rd BD Z BENDING POS ->
AND       M1902F	// DRY RUN
DMOV      D004804 D002352	// R_3rd BD Z ¡Æ¢®¨ùO
DMOV      D004824 D002354	// R_3rd BD Z ¡Æ¡§¨ùO
DMOV      D004846 D002342	// R_3rd BD Z ¢¬nC¡ÍA¡×A¢®
DMOV      D004864 D002344	// R_3rd BD Z ¢¬nC¡Í¨ùO¥ì¥ì
; L109
LOAD NOT  M00600	// EMERGENCY ALARM
AND NOT   D001340.6	// R_3rd BD Z SVD BUSY
AND NOT   D001340.A	// R_3rd BD Z WARNING
AND NOT   D001340.B	// R_3rd BD Z MODULE ERR
AND NOT   D001340.C	// R_3rd BD Z SVD ERR
AND NOT   M02181	// T)R_3rd BD Z JOG-
AND NOT   M02182	// T)R_3rd BD Z JOG+
AND NOT   M02183	// T)R_3rd BD Z SERVO ON
AND NOT   M0318C	// R_3rd BD Z HOME->
AND NOT   M00783	// R_3rd BD Z NOT MV
NOT
OUT       M0168C	// R_3rd BD Z HOLD CUT

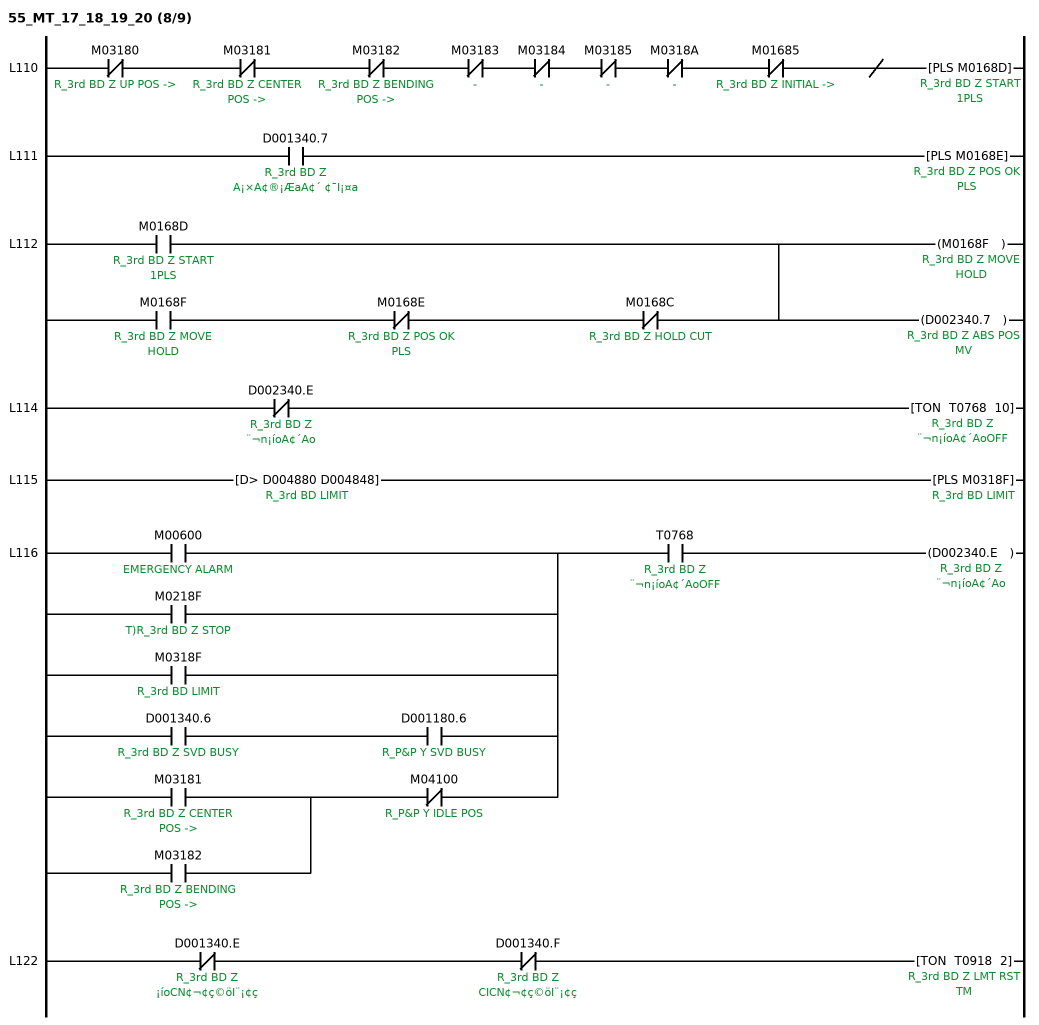
; L110
LOAD NOT  M03180	// R_3rd BD Z UP POS ->
AND NOT   M03181	// R_3rd BD Z CENTER POS ->
AND NOT   M03182	// R_3rd BD Z BENDING POS ->
AND NOT   M03183	// -
AND NOT   M03184	// -
AND NOT   M03185	// -
AND NOT   M0318A	// -
AND NOT   M01685	// R_3rd BD Z INITIAL ->
NOT
OUTP      M0168D	// R_3rd BD Z START 1PLS
; L111
LOAD      D001340.7	// R_3rd BD Z A¡×A¢®¡ÆaA¢´ ¢¯I¡¤a
OUTP      M0168E	// R_3rd BD Z POS OK PLS
; L112
LOAD      M0168D	// R_3rd BD Z START 1PLS
LOAD      M0168F	// R_3rd BD Z MOVE HOLD
AND NOT   M0168E	// R_3rd BD Z POS OK PLS
AND NOT   M0168C	// R_3rd BD Z HOLD CUT
OR LOAD
OUT       M0168F	// R_3rd BD Z MOVE HOLD
OUT       D002340.7	// R_3rd BD Z ABS POS MV
; L114
LOAD NOT  D002340.E	// R_3rd BD Z ¨¬n¡íoA¢´Ao
TON       T0768 10	// R_3rd BD Z ¨¬n¡íoA¢´AoOFF
; L115
LOADD>    D004880 D004848	// R_3rd BD LIMIT
OUTP      M0318F	// R_3rd BD LIMIT
; L116
LOAD      M00600	// EMERGENCY ALARM
OR        M0218F	// T)R_3rd BD Z STOP
OR        M0318F	// R_3rd BD LIMIT
LOAD      D001340.6	// R_3rd BD Z SVD BUSY
AND       D001180.6	// R_P&P Y SVD BUSY
OR LOAD
LOAD      M03181	// R_3rd BD Z CENTER POS ->
OR        M03182	// R_3rd BD Z BENDING POS ->
AND NOT   M04100	// R_P&P Y IDLE POS
OR LOAD
AND       T0768	// R_3rd BD Z ¨¬n¡íoA¢´AoOFF
OUT       D002340.E	// R_3rd BD Z ¨¬n¡íoA¢´Ao
; L122
LOAD NOT  D001340.E	// R_3rd BD Z ¡íoCN¢¬¢ç©öI¨¡¢ç
AND NOT   D001340.F	// R_3rd BD Z CICN¢¬¢ç©öI¨¡¢ç
TON       T0918 2	// R_3rd BD Z LMT RST TM

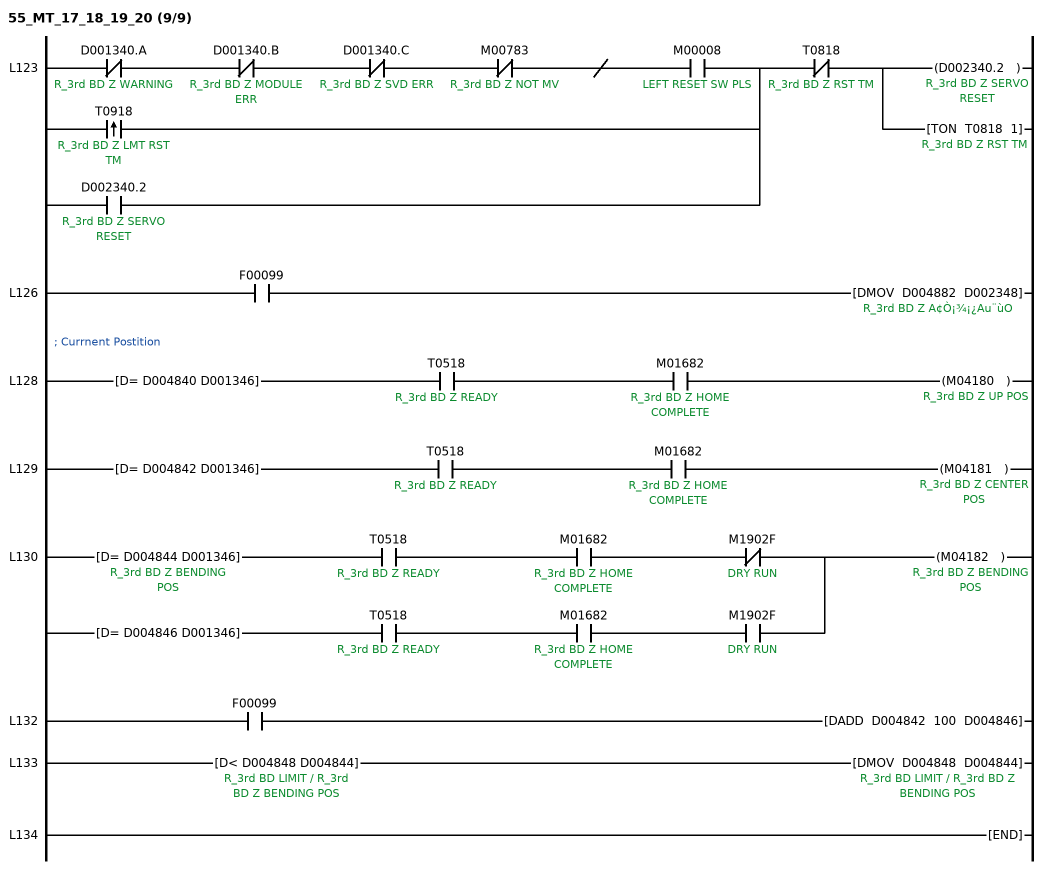
; L123
LOAD NOT  D001340.A	// R_3rd BD Z WARNING
AND NOT   D001340.B	// R_3rd BD Z MODULE ERR
AND NOT   D001340.C	// R_3rd BD Z SVD ERR
AND NOT   M00783	// R_3rd BD Z NOT MV
NOT
AND       M00008	// LEFT RESET SW PLS
ORP       T0918	// R_3rd BD Z LMT RST TM
OR        D002340.2	// R_3rd BD Z SERVO RESET
AND NOT   T0818	// R_3rd BD Z RST TM
OUT       D002340.2	// R_3rd BD Z SERVO RESET
TON       T0818 1	// R_3rd BD Z RST TM
; L126
LOAD      F00099
DMOV      D004882 D002348	// R_3rd BD Z A¢Ò¡¾¡¿Au¨ùO
// Currnent Postition
; L128
LOADD=    D004840 D001346
AND       T0518	// R_3rd BD Z READY
AND       M01682	// R_3rd BD Z HOME COMPLETE
OUT       M04180	// R_3rd BD Z UP POS
; L129
LOADD=    D004842 D001346
AND       T0518	// R_3rd BD Z READY
AND       M01682	// R_3rd BD Z HOME COMPLETE
OUT       M04181	// R_3rd BD Z CENTER POS
; L130
LOADD=    D004844 D001346	// R_3rd BD Z BENDING POS
AND       T0518	// R_3rd BD Z READY
AND       M01682	// R_3rd BD Z HOME COMPLETE
AND NOT   M1902F	// DRY RUN
LOADD=    D004846 D001346
AND       T0518	// R_3rd BD Z READY
AND       M01682	// R_3rd BD Z HOME COMPLETE
AND       M1902F	// DRY RUN
OR LOAD
OUT       M04182	// R_3rd BD Z BENDING POS
; L132
LOAD      F00099
DADD      D004842 100 D004846
; L133
LOADD<    D004848 D004844	// R_3rd BD LIMIT / R_3rd BD Z BENDING POS
DMOV      D004848 D004844	// R_3rd BD LIMIT / R_3rd BD Z BENDING POS
; L134
END

PROGRAM 81_OUTPUT (task: ¨ö¨¬A¥ì CA¡¤I¡¾¡¿¡¤¡Í)

